// TwinCAT 3 PLC project Recipe_Tool
// ProgramVersion: 3.1.0.8
// libraries:
//   Tc2_Standard, * (Beckhoff Automation GmbH)
//   Tc2_System, * (Beckhoff Automation GmbH)
//   Tc3_Interfaces, * (Beckhoff Automation GmbH)
//   Tc3_Module, * (Beckhoff Automation GmbH)
//   Tc3_PLCopen_OpcUa,3.1.1.0,Beckhoff Automation GmbH
//   UML Statechart Types,4.0.0.0,3S - Smart Software Solutions GmbH
// project tree:
//   DUTs/DUTs/Production List/ DUT_SKILL.TcDUT, DUT_TASK.TcDUT, DUT_TASKSTATE.TcDUT
//   DUTs/DUTs/Queue/ DUT_RECIPEORDER.TcDUT, DUT_RECIPE_USERPARAMETERINPUT.TcDUT
//   DUTs/DUTs/RecipeOffer/ DUT_RECIPEOFFER.TcDUT, DUT_RECIPE_USERPARAMETEROUTPUT.TcDUT
//   DUTs/DUT_BASE/ DUT_PARAMETER_INPUT.TcDUT, DUT_PARAMETER_OUTPUT.TcDUT
//   DUTs/ DUT_MODE.TcDUT, DUT_PARAMETER.TcDUT, DUT_RecipeCommand.TcDUT, DUT_RecToolRECIPEOFFER.TcDUT, DUT_STATEVALUES.TcDUT
//   DUTs/DUT_SERVER/ DUT_SERVER_MODULE_INTERFACE.TcDUT, DUT_SERVER_MODULE_INTERFACE_INPUT.TcDUT, DUT_SERVER_MODULE_INTERFACE_OUTPUT.TcDUT, DUT_SERVER_PARAMETERARRAY.TcDUT, DUT_SERVER_PARAMETERINPUTARRAY.TcDUT, DUT_SERVER_PARAMETEROUTPUTARRAY.TcDUT, DUT_SERVER_SKILL.TcDUT, DUT_SERVER_SKILLARRAY.TcDUT, DUT_SERVER_SKILLINPUTARRAY.TcDUT, DUT_SERVER_SKILLOUTPUTARRAY.TcDUT, DUT_SERVER_SKILL_INPUT.TcDUT, DUT_SERVER_SKILL_OUTPUT.TcDUT, DUT_SERVER_STATEVALUEARRAY.TcDUT, DUT_SERVER_TASK.TcDUT
//   GVLs/ GVL.TcGVL, I_O_GVL.TcGVL, OPCConstants.TcGVL
//   / PlcTask.TcTTO
//   POUs/ FB_AddSkill.TcPOU, FB_ExecuteRecipe.TcPOU, FB_INIT_RECIPE.TcPOU, MAIN.TcPOU, Testing.TcPOU
//   POUs/OPC/ FB_OPCServerConnect.TcPOU, FB_ReadReset.TcPOU, FB_ReadRecipeTool.TcPOU, FB_ReadQueue.TcPOU, FB_UpdateRecipeTool.TcPOU, FB_WriteOfferlist.TcPOU, FB_WriteReset.TcPOU, FB_WriteTask.TcPOU, FB_WriteQueue.TcPOU
//   POUs/Recipes/ Recipe_10000_BlankRecipe.TcPOU, Recipe_10001_OneRound.TcPOU, Recipe_10019_DoubleCookieSimu.TcPOU, Recipe_10018_TripleCookiemitTopping.TcPOU, Recipe_10030_HandModule.TcPOU, Recipe_10050_PumpTest.TcPOU, Recipe_10010_transportreserve.TcPOU, Recipe_10011_Skill1337.TcPOU, Recipe_10012_Skill1337_1338_1339.TcPOU, Recipe_10015_eineCookiebitte.TcPOU, Recipe_10013_nSchichten.TcPOU, Recipe_10014_nSchichten4skills.TcPOU, Recipe_10016_CookiemitTopping.TcPOU, Recipe_10017_DoubleCookiemitTopping.TcPOU, Recipe_10051_FreePassion.TcPOU, Recipe_10054_FreePassion_special.TcPOU, Recipe_10052_Orangenschorle.TcPOU, Recipe_10053_911Targa.TcPOU, Recipe_10054_Sixteen.TcPOU, Recipe_10055_Summerday.TcPOU, Recipe_10056_ArcturianSunrise.TcPOU, Recipe_10057_GreenFive.TcPOU, Recipe_10059_Pina_Batida_Lemon.TcPOU, Recipe_10058_RedOne.TcPOU, Recipe_10100_Initialisation.TcPOU, Recipe_11015_DoubleChocoCookie.TcPOU, Recipe_11020_TequilaSunrise.TcPOU
// real-time tasks:
//   TASK PlcTask: cycle T#10ms, priority 20, ADS port 350

CONFIGURATION Recipe_Tool
    RESOURCE PLC ON TwinCAT3
        TASK PlcTask(INTERVAL := T#10ms, PRIORITY := 20);
        PROGRAM MAIN WITH PlcTask : MAIN;
        PROGRAM Testing WITH PlcTask : Testing;
    END_RESOURCE
END_CONFIGURATION

// ---- DUTs/DUTs/Production List/DUT_SKILL.TcDUT
///  Skill variables inside DUT_TASK
TYPE DUT_SKILL :
STRUCT
	///Name assigned for the process tool
	AssignedModuleName: STRING(80);
	///ID assigned for the process tool
	AssignedModuleID: UINT;
	///Position assigned for the process tool
	AssignedModulePosition: LREAL;
	///Free to use = TRUE, busy to use =FALSE
	Dummy: BOOL := TRUE;
	///Identification number of the skill
	ID: UINT;
	///Name of the skill
	Name: STRING(80);
	///Range of parameters
	Parameter: ARRAY[0..ParameterCnt] OF DUT_PARAMETER;
END_STRUCT
END_TYPE

// ---- DUTs/DUTs/Production List/DUT_TASK.TcDUT
TYPE DUT_TASK :
STRUCT
	///Name of the Task
	Name: STRING(80);
	///Free to use = TRUE, busy to use =FALSE
	Dummy: BOOL := TRUE;
	///Identification number of the Task
	TaskID: INT;
	///Identification number of the Recipe
	RecipeID: INT;
	///Range of Skill in the TASK
	Skill: ARRAY[0..TaskSkillCnt] OF DUT_SKILL;
	///When occurs the action
	Timestamp: STRING(80);
	///State of the TASK e.g (unassigned, assigned, waitingForSkillReady, inProgress, done, aborted, error)
	State: DUT_TASKSTATE := 0;
END_STRUCT
END_TYPE

// ---- DUTs/DUTs/Production List/DUT_TASKSTATE.TcDUT
TYPE DUT_TASKSTATE :
(
	Unassigned := 0,
	///Assigned := 1,
	WaitingForSkillReady := 1,
	InProgress := 2,
	Done := 3,
	Aborted := 4,
	Error := 5
);
END_TYPE

// ---- DUTs/DUTs/Queue/DUT_RECIPEORDER.TcDUT
TYPE DUT_RECIPEORDER :
STRUCT
	Locked: BOOL;
	Pending: BOOL;
	///corelating to the offered recipes#
	RecipeID: INT;
	///continious numbering
	TaskID: INT;
	Name: STRING(80);
	Description: STRING(255);
	UserParameter: ARRAY[0..UserParameterCnt] OF DUT_RECIPE_USERPARAMETERINPUT;
END_STRUCT
END_TYPE

// ---- DUTs/DUTs/Queue/DUT_RECIPE_USERPARAMETERINPUT.TcDUT
TYPE DUT_RECIPE_USERPARAMETERINPUT :
STRUCT
	Value: REAL;
END_STRUCT
END_TYPE

// ---- DUTs/DUTs/RecipeOffer/DUT_RECIPEOFFER.TcDUT
TYPE DUT_RECIPEOFFER :
STRUCT
	Dummy: BOOL := TRUE;
	Name: STRING(80) := 'e.g. Product x';
	RecipeID: INT;
	Description: STRING(255) := '%Description of the Recipe e.g. "a recipe, that produces a product with feature x"';
	UserParameter: ARRAY[0..UserParameterCnt] OF DUT_RECIPE_USERPARAMETEROUTPUT;
END_STRUCT
END_TYPE

// ---- DUTs/DUTs/RecipeOffer/DUT_RECIPE_USERPARAMETEROUTPUT.TcDUT
TYPE DUT_RECIPE_USERPARAMETEROUTPUT :
STRUCT
	Dummy: BOOL := TRUE;
	Name: STRING(80);
	Description: STRING(80);
	Unit: STRING(80);
	MinValue: LREAL;
	MaxValue: LREAL;
	Default: LREAL;
	Step: LREAL;
END_STRUCT
END_TYPE

// ---- DUTs/DUT_BASE/DUT_PARAMETER_INPUT.TcDUT
TYPE DUT_PARAMETER_INPUT :
STRUCT
	///Value of the parameter 
	Value: LREAL;
	///Possibility to a string value depending on the parameter
	StringValue: STRING[80];
END_STRUCT
END_TYPE

// ---- DUTs/DUT_BASE/DUT_PARAMETER_OUTPUT.TcDUT
TYPE DUT_PARAMETER_OUTPUT :
STRUCT
	///Free to use = TRUE, busy to use =FALSE
	Dummy: BOOL := TRUE;
	///ID of the parameter
	ID: UINT;
	///Name of the parameter
	Name: STRING[80];
	///Unit of the parameter
	Unit: STRING[80];
	///Optional parameter
	Required: BOOL;
	///Default parameter to work
	Default: LREAL;
	///Minimum value of the parameter
	MinValue: LREAL;
	///Maximum value of the parameter
	MaxValue: LREAL;
END_STRUCT
END_TYPE

// ---- DUTs/DUT_MODE.TcDUT
/// MODE to run (inside of MODULE_INTERFACE_INPUT)
TYPE DUT_MODE :
(
	///Initialitzation number mode
	Init := 0,
	///Automatic number mode
	Auto := 1,
	///Manual number mode
	Manual := 2,
	Reset := 3
);
END_TYPE

// ---- DUTs/DUT_PARAMETER.TcDUT
TYPE DUT_PARAMETER :
STRUCT
	///Free to use = TRUE, busy to use =FALSE
	Dummy: BOOL := TRUE;
	///ID of the parameter
	ID: UINT;
	///Name of the parameter
	Name: STRING[80];
	///Unit of the parameter (mm,L,...)
	Unit: STRING[80];
	///Optional parameter
	Required: BOOL;
	///Default parameter to work
	Default: LREAL;
	///Minimum value of the parameter
	MinValue: LREAL;
	///Maximum value of the parameter
	MaxValue: LREAL;
	///Actual Value
	Value: LREAL;
	///StringValue
	StringValue: STRING[80];
END_STRUCT
END_TYPE

// ---- DUTs/DUT_RecipeCommand.TcDUT
TYPE DUT_RecipeCommand :
STRUCT
	SkillID: INT;
	SkillName: STRING(80);
	Quantity: LREAL;
END_STRUCT
END_TYPE

// ---- DUTs/DUT_RecToolRECIPEOFFER.TcDUT
TYPE DUT_RecToolRECIPEOFFER :
STRUCT
	Dummy:			BOOL := TRUE;
	Name:			STRING[80]:= 'e.g. Product x';
	RecipeID:		INT;
	Description:	STRING[80]:= '%Description of the Recipe e.g. "a recipe, that produces a product with feature x"';
	UserParameter:  DUT_RECIPE_USERPARAMETEROUTPUT;
END_STRUCT
END_TYPE

// ---- DUTs/DUT_SERVER/DUT_SERVER_MODULE_INTERFACE.TcDUT
/// MODULE INTERFACE INPUT AND OUTPUT 
TYPE DUT_SERVER_MODULE_INTERFACE :
STRUCT
	///Information that the module reads
	Input: DUT_SERVER_MODULE_INTERFACE_INPUT;
	///Information that the module write
	Output: DUT_SERVER_MODULE_INTERFACE_OUTPUT;
END_STRUCT
END_TYPE

// ---- DUTs/DUT_SERVER/DUT_SERVER_MODULE_INTERFACE_INPUT.TcDUT
TYPE DUT_SERVER_MODULE_INTERFACE_INPUT :
STRUCT
	///Mode to run (init,auto,manual,..)
	Mode: DUT_MODE;
	///check if the modules is alive
	ConnectionTestInput: BOOL;
	///Modules get their position
	PositionInput: LREAL;
	///Update data= TRUE, No updatedata=FALSE
	Watchbit: BOOL;
	///Emergency stop
	EmergencyStop: BOOL;
	///Range of INPUT skills
	SkillInput: DUT_SERVER_SKILLINPUTARRAY;
END_STRUCT
END_TYPE

// ---- DUTs/DUT_SERVER/DUT_SERVER_MODULE_INTERFACE_OUTPUT.TcDUT
TYPE DUT_SERVER_MODULE_INTERFACE_OUTPUT :
STRUCT
	///Free to use = TRUE, busy to use =FALSE
	Dummy: BOOL := TRUE;
	///Individual name of the module
	Name: STRING[80];
	///Identification number of module
	ID: UINT;
	///IP address
	IP: STRING[80];
	///Show if the module is in Standby or not
	Idle: BOOL;
	///Show if the module is connected
	Connected: BOOL;
	///Feedback with conection test input
	ConnectionTestOutput: BOOL;
	///Show if the system has error when=TRUE
	Error: BOOL;
	///Identification number of the error
	ErrorID: UINT;
	///Description of the error
	ErrorDescription: STRING[80];
	///Description of the current task
	CurrentTaskDescription: STRING[80];
	///Position of the sensor
	PositionSensor: BOOL;
	///Range of OUTPUT skills
	SkillOutput: DUT_SERVER_SKILLOUTPUTARRAY;
	///Range of state values
	StateValue: DUT_SERVER_STATEVALUEARRAY;
END_STRUCT
END_TYPE

// ---- DUTs/DUT_SERVER/DUT_SERVER_PARAMETERARRAY.TcDUT
TYPE DUT_SERVER_PARAMETERARRAY :
STRUCT
	Parameter0 : DUT_PARAMETER;
	Parameter1 : DUT_PARAMETER;
	Parameter2 : DUT_PARAMETER;
	Parameter3 : DUT_PARAMETER;
	Parameter4 : DUT_PARAMETER;
	Parameter5 : DUT_PARAMETER;
	
END_STRUCT
END_TYPE

// ---- DUTs/DUT_SERVER/DUT_SERVER_PARAMETERINPUTARRAY.TcDUT
TYPE DUT_SERVER_PARAMETERINPUTARRAY :
STRUCT
		Parameterinput0	: DUT_PARAMETER_INPUT;
	Parameterinput1	: DUT_PARAMETER_INPUT;
	Parameterinput2	: DUT_PARAMETER_INPUT;
	Parameterinput3	: DUT_PARAMETER_INPUT;
	Parameterinput4	: DUT_PARAMETER_INPUT;
	Parameterinput5	: DUT_PARAMETER_INPUT;
END_STRUCT
END_TYPE

// ---- DUTs/DUT_SERVER/DUT_SERVER_PARAMETEROUTPUTARRAY.TcDUT
TYPE DUT_SERVER_PARAMETEROUTPUTARRAY :
STRUCT
	ParameterOutput0	: DUT_PARAMETER_OUTPUT;
	ParameterOutput1	: DUT_PARAMETER_OUTPUT;
	ParameterOutput2	: DUT_PARAMETER_OUTPUT;
	ParameterOutput3	: DUT_PARAMETER_OUTPUT;
	ParameterOutput4	: DUT_PARAMETER_OUTPUT;
	ParameterOutput5	: DUT_PARAMETER_OUTPUT;
END_STRUCT
END_TYPE

// ---- DUTs/DUT_SERVER/DUT_SERVER_SKILL.TcDUT
///  Skill variables inside DUT_TASK
TYPE DUT_SERVER_SKILL :
STRUCT
	///Name assigned for the process tool
	AssignedModuleName: STRING[80];
	///ID assigned for the process tool
	AssignedModuleID: UINT;
	///Position assigned for the process tool
	AssignedModulePosition: UINT;
	///Free to use = TRUE, busy to use =FALSE
	Dummy: BOOL := TRUE;
	///Identification number of the skill
	ID: UINT;
	///Name of the skill
	Name: STRING[80];
	///Range of parameters
	Parameter : DUT_SERVER_PARAMETERARRAY;
END_STRUCT
END_TYPE

// ---- DUTs/DUT_SERVER/DUT_SERVER_SKILLARRAY.TcDUT
TYPE DUT_SERVER_SKILLARRAY :
STRUCT
	Skill0 : DUT_SERVER_SKILL;
	Skill1 : DUT_SERVER_SKILL;
	Skill2 : DUT_SERVER_SKILL;
	Skill3 : DUT_SERVER_SKILL;
	Skill4 : DUT_SERVER_SKILL;
	Skill5 : DUT_SERVER_SKILL;
	Skill6 : DUT_SERVER_SKILL;
	Skill7 : DUT_SERVER_SKILL;
	Skill8 : DUT_SERVER_SKILL;
	Skill9 : DUT_SERVER_SKILL;
	Skill10 : DUT_SERVER_SKILL;
	Skill11 : DUT_SERVER_SKILL;
	Skill12 : DUT_SERVER_SKILL;
	Skill13 : DUT_SERVER_SKILL;
	Skill14 : DUT_SERVER_SKILL;
	Skill15 : DUT_SERVER_SKILL;
	Skill16 : DUT_SERVER_SKILL;
	Skill17 : DUT_SERVER_SKILL;
	Skill18 : DUT_SERVER_SKILL;
	Skill19 : DUT_SERVER_SKILL;	
	Skill20 : DUT_SERVER_SKILL;
	Skill21 : DUT_SERVER_SKILL;
	Skill22 : DUT_SERVER_SKILL;
	Skill23 : DUT_SERVER_SKILL;
	Skill24 : DUT_SERVER_SKILL;
	Skill25 : DUT_SERVER_SKILL;
	Skill26 : DUT_SERVER_SKILL;
	Skill27 : DUT_SERVER_SKILL;
	Skill28 : DUT_SERVER_SKILL;
	Skill29 : DUT_SERVER_SKILL;
	Skill30 : DUT_SERVER_SKILL;
	Skill31 : DUT_SERVER_SKILL;
	Skill32 : DUT_SERVER_SKILL;
	Skill33 : DUT_SERVER_SKILL;
	Skill34 : DUT_SERVER_SKILL;
	Skill35 : DUT_SERVER_SKILL;
	Skill36 : DUT_SERVER_SKILL;
	Skill37 : DUT_SERVER_SKILL;
	Skill38 : DUT_SERVER_SKILL;
	Skill39 : DUT_SERVER_SKILL;
	Skill40 : DUT_SERVER_SKILL;
	Skill41 : DUT_SERVER_SKILL;
	Skill42 : DUT_SERVER_SKILL;
	Skill43 : DUT_SERVER_SKILL;
	Skill44 : DUT_SERVER_SKILL;
	Skill45 : DUT_SERVER_SKILL;
	Skill46 : DUT_SERVER_SKILL;
	Skill47 : DUT_SERVER_SKILL;
	Skill48 : DUT_SERVER_SKILL;
	Skill49 : DUT_SERVER_SKILL;
	Skill50 : DUT_SERVER_SKILL;
END_STRUCT
END_TYPE

// ---- DUTs/DUT_SERVER/DUT_SERVER_SKILLINPUTARRAY.TcDUT
TYPE DUT_SERVER_SKILLINPUTARRAY :
STRUCT
	SkillInput0 : DUT_SERVER_SKILL_INPUT;
	SkillInput1 : DUT_SERVER_SKILL_INPUT;
	SkillInput2 : DUT_SERVER_SKILL_INPUT;
	SkillInput3 : DUT_SERVER_SKILL_INPUT;
	SkillInput4 : DUT_SERVER_SKILL_INPUT;
	SkillInput5 : DUT_SERVER_SKILL_INPUT;
	SkillInput6 : DUT_SERVER_SKILL_INPUT;
	SkillInput7 : DUT_SERVER_SKILL_INPUT;
	SkillInput8 : DUT_SERVER_SKILL_INPUT;
	SkillInput9 : DUT_SERVER_SKILL_INPUT;
	SkillInput10 : DUT_SERVER_SKILL_INPUT;
	SkillInput11 : DUT_SERVER_SKILL_INPUT;
	SkillInput12 : DUT_SERVER_SKILL_INPUT;
	SkillInput13 : DUT_SERVER_SKILL_INPUT;
	SkillInput14 : DUT_SERVER_SKILL_INPUT;
	SkillInput15 : DUT_SERVER_SKILL_INPUT;
END_STRUCT
END_TYPE

// ---- DUTs/DUT_SERVER/DUT_SERVER_SKILLOUTPUTARRAY.TcDUT
TYPE DUT_SERVER_SKILLOUTPUTARRAY :
STRUCT
		SkillOutput0	: DUT_SERVER_SKILL_OUTPUT;
	SkillOutput1	: DUT_SERVER_SKILL_OUTPUT;
	SkillOutput2	: DUT_SERVER_SKILL_OUTPUT;
	SkillOutput3	: DUT_SERVER_SKILL_OUTPUT;
	SkillOutput4	: DUT_SERVER_SKILL_OUTPUT;
	SkillOutput5	: DUT_SERVER_SKILL_OUTPUT;
	SkillOutput6	: DUT_SERVER_SKILL_OUTPUT;
	SkillOutput7	: DUT_SERVER_SKILL_OUTPUT;
	SkillOutput8	: DUT_SERVER_SKILL_OUTPUT;
	SkillOutput9	: DUT_SERVER_SKILL_OUTPUT;
	SkillOutput10	: DUT_SERVER_SKILL_OUTPUT;
	SkillOutput11	: DUT_SERVER_SKILL_OUTPUT;
	SkillOutput12	: DUT_SERVER_SKILL_OUTPUT;
	SkillOutput13	: DUT_SERVER_SKILL_OUTPUT;
	SkillOutput14	: DUT_SERVER_SKILL_OUTPUT;
	SkillOutput15	: DUT_SERVER_SKILL_OUTPUT;
END_STRUCT
END_TYPE

// ---- DUTs/DUT_SERVER/DUT_SERVER_SKILL_INPUT.TcDUT
TYPE DUT_SERVER_SKILL_INPUT :
STRUCT
	///Range of parameters
	ParameterInput: DUT_SERVER_PARAMETERINPUTARRAY;
	///Start process
	Execute: BOOL;
END_STRUCT
END_TYPE

// ---- DUTs/DUT_SERVER/DUT_SERVER_SKILL_OUTPUT.TcDUT
TYPE DUT_SERVER_SKILL_OUTPUT :
STRUCT
	///Free to use = TRUE, busy to use =FALSE
	Dummy: BOOL := TRUE;
	///Identification number of skill
	ID: UINT;
	///indentfication name of skill
	Name: STRING[80];
	///Skill activated
	Activated: BOOL;
	///Ready to do skill
	Ready: BOOL;
	///Skill in process
	Busy: BOOL;
	///Skill finish
	Done: BOOL;
	///Error in system
	Error: BOOL;
	///Range of parameters
	ParameterOutput: DUT_SERVER_PARAMETEROUTPUTARRAY;
END_STRUCT
END_TYPE

// ---- DUTs/DUT_SERVER/DUT_SERVER_STATEVALUEARRAY.TcDUT
TYPE DUT_SERVER_STATEVALUEARRAY :
STRUCT
		Statevalue0	: DUT_STATEVALUES;
	Statevalue1	: DUT_STATEVALUES;
	Statevalue2	: DUT_STATEVALUES;
	Statevalue3	: DUT_STATEVALUES;
	Statevalue4	: DUT_STATEVALUES;
	Statevalue5	: DUT_STATEVALUES;
	Statevalue6	: DUT_STATEVALUES;
	Statevalue7	: DUT_STATEVALUES;
	Statevalue8	: DUT_STATEVALUES;
	Statevalue9	: DUT_STATEVALUES;
	Statevalue10	: DUT_STATEVALUES;
END_STRUCT
END_TYPE

// ---- DUTs/DUT_SERVER/DUT_SERVER_TASK.TcDUT
TYPE DUT_SERVER_TASK :
STRUCT
	///Name of the Task
	Name: STRING[80];
	///Free to use = TRUE, busy to use =FALSE
	Dummy: BOOL := TRUE;
	///Identification number of the Task
	TaskID: INT;
	///Identification number of the Recipe
	RecipeID: INT;
	///Range of Skill in the TASK
	Skill: DUT_SERVER_SKILLARRAY;
	///When occurs the action
	Timestamp: STRING[80];
	///State of the TASK e.g (unassigned, assigned, waitingForSkillReady, inProgress, done, aborted, error)
	State: DUT_TASKSTATE;
END_STRUCT
END_TYPE

// ---- DUTs/DUT_STATEVALUES.TcDUT
TYPE DUT_STATEVALUES :
STRUCT
	Dummy:			BOOL := TRUE;				(*Free to use = TRUE, busy to use =FALSE*)
	Value:			LREAL;						(*Value of the State*)
	Name:			STRING[80];						(*Name of the state*)
	Description:	STRING[80];				(*Description of the state*)
	Unit:			STRING[80];						(*Unit of the state ()*)
END_STRUCT
END_TYPE

// ---- GVLs/GVL.TcGVL
VAR_GLOBAL
	ExecuteSkill	: FB_AddSkill;
	TempTask		: DUT_TASK;
	EmptyTask		: DUT_TASK;
	EmptyQueue		: DUT_RECIPEORDER;
	
	ZCremeModuleCalibration		: LREAL := 0;	
	ZCremeModule				: LREAL	:= 101;
	
	
	ZCocktailModuleCalibration 	: LREAL := 0;
	ZCocktailModule				: LREAL := 20;
	
	ZCookieModuleCalibration	: LREAL := 0;
	ZCookieModule				: LREAL := 90.0;
	
	ZInputOutput				: LREAL := 109;
	
	
	
	cookiethickness				: LREAL := 5.0;
	toppingthickness			: LREAL := 1.0;
	
	preasureheight				: LREAL := 30.0;
	ClearTaskList				: BOOL;	
	ClearManual					: BOOL;
END_VAR

// ---- GVLs/I_O_GVL.TcGVL
VAR_GLOBAL
// Inputs:

Queue	: DUT_RECIPEORDER;

//Outputs:

Offer	: ARRAY [0..OfferCnt] OF DUT_RECIPEOFFER;

// ProductionList

Task	: ARRAY [0..TaskCnt] OF DUT_TASK;
END_VAR

// ---- GVLs/OPCConstants.TcGVL
VAR_GLOBAL CONSTANT
	///Maximum number of skillparameters:
	ParameterCnt: INT := 5;
	///Maximum number of skills per Module:
	SkillCnt: INT := 15;
	///Maximum number of Statevalues of one Module:
	StateCnt: INT := 10;
	///Maximum number of modules:
	ModuleCnt: INT := 10;
	///Maximum number of Tasks in Production List:
	TaskCnt: INT := 30;
	///Maximum number  of offered recipes:
	OfferCnt: INT := 30;
	///Maximum number of Orders in Queue:
	OrderCnt: INT := 5;
	///Number of user set parameters per recipe:
	UserParameterCnt: INT := 5;
	///Number of skills per task:
	TaskSkillCnt: INT := 50;
	
	
END_VAR

// ---- POUs/MAIN.TcPOU
PROGRAM MAIN
VAR
	
		
	state	: INT := -40;	
	i		: INT;
	connectcounter	: INT;
	TaskListPosition: INT := -1;
	TaskListPositionString	: STRING[80];
	Tempstring		: STRING[80];
	//FB Instances
	TranslateRecipe	: FB_ExecuteRecipe;
	fbInitOffers	: FB_INIT_RECIPE;	
	//OPC Instances:
	//fbOPCUpdate		: FB_UpdateRecipeTool;
	fbReadReset			: FB_ReadReset;
	fbWriteReset		: FB_WriteReset;
	fbOPCConnect		: FB_OPCServerConnect;
	fbWriteOffers		: FB_WriteOfferlist;
	fbReadQueue			: FB_ReadQueue;
	fbWriteTask			: FB_WriteTask;
	fbWriteQueue		: FB_WriteQueue;
	fbDisconnect		: UA_Disconnect;
	NamespaceIndex		: UINT;
	ConnectionHdl		: DWORD;
	TaskIdentifier		: STRING[80];
	sizeofRecipfOFfer	: INT;
	ClearOrder			: DUT_RECIPEORDER;
	ToolTimeout			: TON;
	Trigger				: R_TRIG;
	TriggerState		: INT;
	ResetReadTimer		: TON;
	
END_VAR


CASE state OF
	-40: //Initialate Recipe Offer List
		fbInitOffers(Execute := TRUE);
		ToolTimeout(IN := FALSE);
		IF fbInitOffers.Done THEN
			state := -30;
		END_IF
	-35: fbDisconnect(ConnectionHdl := ConnectionHdl,Timeout := T#4S, Execute := FALSE);
		state := -34;
	-34: fbDisconnect(ConnectionHdl := ConnectionHdl,Timeout := T#4s, Execute := TRUE);
		IF nOT fbDisconnect.busy  THEN
			state := -30;
		END_IF
		
	
	-30: fbOPCConnect(
						ServerUrl:= 'opc.tcp://192.168.42.42:4840',//'opc.tcp://192.168.192.116:4840', 
						NamespaceUri:= 'PLC1', 
						ClientName:= 'RecipeTool', 
						execute:= TRUE, 
						ConnectHdl=> ConnectionHdl, 
						Namespaceindex=> NamespaceIndex, 
						busy=> , 
						done=> , 
						error=> );
		IF fbOPCConnect.done THEN
			state := -15;
		END_IF
					
		
	
	
	
	-15: // OPC WRITE 
		fbWriteOffers(
						WriteIdentifier:= 'MI5.Recipe', 
						NamespaceIndex:= NamespaceIndex, 
						ConnectionHdl:= ConnectionHdl, 
						execute:= TRUE, 
						WriteData:= Offer, 
						done=> , 
						busy=> , 
						error=> );
		IF fbWriteOffers.done THEN
			state := -10;
		END_IF

	
	-10: //INIT DONE
		TranslateRecipe.InitDone := TRUE;
		state := 0;
	
	
	
	 0:		// Waiting for new Order
	 	IF NOT Testing.NoOPC THEN
	 		fbReadQueue(
						ReadIdentifier:= 'MI5.Order[0]', 
						NamespaceIndex:= NamespaceIndex, 
						ConnectionHdl:= ConnectionHdl, 
						execute:= TRUE, 
						ReadData=> Queue, 
						done=> , 
						busy=> , 
						error=> );
			IF fbReadQueue.done THEN
				state := 1;
			END_IF
		ELSE
			state := 5;
		END_IF
		
	1:	
		IF NOT Testing.NoOPC THEN
				fbReadQueue(
							ReadIdentifier:= 'MI5.Order[0]', 
							NamespaceIndex:= NamespaceIndex, 
							ConnectionHdl:= ConnectionHdl, 
							execute:= TRUE, 
							ReadData=> Queue, 
							done=> , 
							busy=> , 
							error=> );
				Trigger(CLK := fbReadQueue.done);
				ToolTimeout(IN := NOT Trigger.Q);
							
				IF Queue.Pending THEN
					state := 10;
					TaskListPosition := TaskListPosition +1;
						//Reset bei Overflow
						IF TaskListPosition > 29 THEN
							TaskListPosition := 0;
						END_IF
				END_IF		
		ELSE
			state := 5;
		END_IF
	 5:
		IF Queue.Pending THEN
			state := 10;
			TaskListPosition := TaskListPosition +1;
				//Reset bei Overflow
				IF TaskListPosition > 29 THEN
					TaskListPosition := 0;
				END_IF
		END_IF
	 	
	 
	10: state := 20;
		
		
	20: //Translate corresponding offer to TempTask
		TranslateRecipe(Order:= Queue, Done=> , Execute := TRUE);
		
		IF TranslateRecipe.Done THEN
			state := 21;//21;
			ExecuteSkill.TargetSkillNo := 0;
		END_IF
		
		
		//todo quatsch recipe IDs abfangen? return an HMI
	21: TempTask.Name := Queue.Name;
		TempTask.Dummy := FALSE;
		TempTask.RecipeID := Queue.RecipeID;
		TempTask.TaskID := Queue.TaskID;
		TempTask.State := 1;
		TempTask.Timestamp := 'mytimestamp';
		state := 25;
		
			
	25: //Parse write identifier
		TaskListPositionString := INT_TO_STRING(TaskListPosition);
		Tempstring := CONCAT(STR1:= 'MI5.ProductionList[', STR2:= TaskListPositionString );
		
		TaskIdentifier := CONCAT(STR1:= Tempstring, STR2:=']' );
		state := 30;	
	30: // Copy to local Production List
		fbWriteTask(
					WriteIdentifier:= TaskIdentifier, 
					NamespaceIndex:= NamespaceIndex, 
					ConnectionHdl:= ConnectionHdl, 
					execute:= TRUE, 
					WriteData:= TempTask, 
					done=> , 
					busy=> , 
					error=> );
		IF fbWriteTask.done THEN
		//
		state := 40;
		END_IF		
	

	40:  // free Queue Slot
		TempTask				:= EmptyTask;
		IF NOT Testing.NoOPC THEN
			fbWriteQueue(
				WriteIdentifier:= 'MI5.Order[0]', 
				NamespaceIndex:= NamespaceIndex, 
				ConnectionHdl:= ConnectionHdl, 
				execute:= TRUE, 
				WriteData:= , 
				done=> , 
				busy=> , 
				error=> );
			IF fbWriteQueue.done THEN
			state := 0;
			END_IF
		ELSE
			Queue.Pending := FALSE;
			state := 0;
		END_IF
	
	
		
		
		
	125: //Parse write identifier
		TaskListPositionString := INT_TO_STRING(i);
		Tempstring := CONCAT(STR1:= 'MI5.ProductionList[', STR2:= TaskListPositionString );
		
		TaskIdentifier := CONCAT(STR1:= Tempstring, STR2:=']' );
		state := 130;	
	130: // Copy to local Production List
		fbWriteTask(
					WriteIdentifier:= TaskIdentifier, 
					NamespaceIndex:= NamespaceIndex, 
					ConnectionHdl:= ConnectionHdl, 
					execute:= TRUE, 
					WriteData:= EmptyTask, 
					done=> , 
					busy=> , 
					error=> );
		IF fbWriteTask.done THEN
			IF  i <TaskCnt  THEN
				i := i +1;
				state := 125;
			ELSE
				state := -30;
				i := -1;
			END_IF
		
		END_IF		
		
		
END_CASE



sizeofRecipfOFfer := SIZEOF(DUT_RecipeOffer);

//TImerout:
ToolTimeout(IN := TRUE, PT := T#20S);


//stateänderungsüberprüfung
IF NOT (state  = triggerstate) THEN
	ToolTimeout(IN:= FALSE);
END_IF
triggerstate := state;


IF ToolTimeout.Q THEN
	connectcounter	:= connectcounter +1;
	state := -35;
	ToolTimeout(IN:= FALSE);
	fbOPCConnect	(execute := FALSE);			
	fbWriteOffers	(execute := FALSE);		
	fbReadQueue		(execute := FALSE);			
	fbWriteTask		(execute := FALSE);			
	fbWriteQueue	(execute := FALSE);		
	
END_IF

ResetReadTimer(IN := TRUE, PT := T#3S);
IF ResetReadTimer.Q THEN
	ResetReadTimer(IN := FALSE);
	ResetReadTimer(IN := TRUE);
	fbReadReset.execute := TRUE;
END_IF
fbReadReset(		ReadIdentifier:= 'MI5.ClearTaskList', 
					NamespaceIndex:= NamespaceIndex, 
					ConnectionHdl:= ConnectionHdl, 
					execute:= , 
					ReadData=> ClearTaskList, 
					done=> , 
					busy=> , 
					error=> 
				);

					
IF ClearTaskList OR ClearManual THEN
	i := 0;
	ClearManual := FALSE;
	Tasklistposition := -1;
	fbWriteReset(	WriteIdentifier := 'MI5.ClearTaskList',
					NamespaceIndex := NamespaceIndex, 
					ConnectionHdl := ConnectionHdl, 
					WriteData := FALSE,
					Execute		:= TRUE);
	IF fbWriteReset.done THEN
		state := 125;
	END_IF
	
END_IF

END_PROGRAM

// ---- POUs/FB_ExecuteRecipe.TcPOU
FUNCTION_BLOCK FB_ExecuteRecipe
VAR_INPUT
	Order			: 	DUT_RECIPEORDER;
	Execute			: 	BOOL;
	InitDone		: 	BOOL;
END_VAR
VAR_OUTPUT
	Done	:	BOOL;
	NotAvailable: BOOL;
	RecipeInfo	: DUT_RECIPEOFFER;
END_VAR
VAR
		BriefcaseConfig	: BOOL := TRUE;
		i			: INT;
		Recipe10001 : Recipe_10001_OneRound;
		Recipe10010 : Recipe_10010_transportreserve;
		
		
		//Recipe11020	: Recipe_11020_TequilaSunrise;
		Recipe10000 : Recipe_10000_BlankRecipe;
		//Recipe10013 : Recipe_10013_nSchichten;
		//Recipe10014 : Recipe_10014_nSchichten4skills;
		//Recipe20014	: Recipe_20014_chocoCookie;
		Recipe10011: Recipe_10011_Skill1337;
		//Recipe10012: Recipe_10012_Skill1337_1338_1339;
		//Recipe10015: Recipe_10015_eineCookiebitte;
		//Recipe10016: Recipe_10016_CookiemitTopping;
		Recipe10017: Recipe_10017_DoubleCookiemitTopping;
		//Recipe10018: Recipe_10018_TripleCookiemitTopping;
		Recipe10019: Recipe_10019_DoubleCookieSimu;
		//Recipe10050: Recipe_10050_PumpTest;
		Recipe10051: Recipe_10051_FreePassion;
		//Recipe10052: Recipe_10052_Orangenschorle;
		Recipe10053: Recipe_10053_911Targa;
		//Recipe10054: Recipe_10054_FreePassion_special;
		Recipe10055: Recipe_10055_Summerday;
		Recipe10056: Recipe_10056_ArcturianSunrise;
		Recipe10057: Recipe_10057_GreenFive;
		//Recipe10058: Recipe_10058_RedOne;
		//Recipe10059: Recipe_10059_Pina_Batida_Lemon;
		
END_VAR





IF Execute THEN
	Done := FALSE;
	NotAvailable := FALSE;
	
	CASE Order.RecipeID OF
		
		(*10000: Recipe10000 (Execute := InitDone,Order := order,RecipeInfo => RecipeInfo);
				
				IF Recipe10000.RecipeDone THEN
					Done := TRUE;
					Execute := FALSE;
					Recipe10000(execute := FALSE);
					
					
				END_IF
		*)		
		
		10001: Recipe10001 (Execute := InitDone,Order := order,RecipeInfo => RecipeInfo);
				
				IF Recipe10001.RecipeDone THEN
					Done := TRUE;
					Execute := FALSE;
					Recipe10001(execute := FALSE);
										
				END_IF	
				
		10010: Recipe10010 (Execute := InitDone,Order := order,RecipeInfo => RecipeInfo);
				
				IF Recipe10010.RecipeDone THEN
					Done := TRUE;
					Execute := FALSE;
					Recipe10010(execute := FALSE);
										
				END_IF
		10011: Recipe10011 (Execute := InitDone,Order := order,RecipeInfo => RecipeInfo);
				
				IF Recipe10011.RecipeDone THEN
					Done := TRUE;
					Execute := FALSE;
					Recipe10011(execute := FALSE);
										
				END_IF
				
		(*10012: Recipe10012 (Execute := InitDone,Order := order,RecipeInfo => RecipeInfo);
				
				IF Recipe10012.RecipeDone THEN
					Done := TRUE;
					Execute := FALSE;
					Recipe10012(execute := FALSE);
										
				END_IF
		*)
		(*
10013: Recipe10013 (Execute := InitDone,Order := order,RecipeInfo => RecipeInfo);
				
				IF Recipe10013.RecipeDone THEN
					Done := TRUE;
					Execute := FALSE;
					Recipe10013(execute := FALSE);
										
				END_IF
				*)
		(*10014: Recipe10014 (Execute := InitDone,Order := order,RecipeInfo => RecipeInfo);
				
				IF Recipe10014.RecipeDone THEN
					Done := TRUE;
					Execute := FALSE;
					Recipe10014(execute := FALSE);
										
				END_IF*)
		(*10015: Recipe10015 (Execute := InitDone,Order := order,RecipeInfo => RecipeInfo);
				
				IF Recipe10015.RecipeDone THEN
					Done := TRUE;
					Execute := FALSE;
					Recipe10015(execute := FALSE);
										
				END_IF
		*)
		
		(*
		10016: Recipe10016 (Execute := InitDone,Order := order,RecipeInfo => RecipeInfo);
				
				IF Recipe10016.RecipeDone THEN
					Done := TRUE;
					Execute := FALSE;
					Recipe10016(execute := FALSE);
										
				END_IF
				*)
				
		10017: Recipe10017 (Execute := InitDone,Order := order,RecipeInfo => RecipeInfo);
				
				IF Recipe10017.RecipeDone THEN
					Done := TRUE;
					Execute := FALSE;
					Recipe10017(execute := FALSE);
										
				END_IF	
		(*10018: Recipe10018 (Execute := InitDone,Order := order,RecipeInfo => RecipeInfo);
				
				IF Recipe10018.RecipeDone THEN
					Done := TRUE;
					Execute := FALSE;
					Recipe10018(execute := FALSE);
										
				END_IF		
			*)	
		10019: Recipe10019 (Execute := InitDone,Order := order,RecipeInfo => RecipeInfo);
				
				IF Recipe10019.RecipeDone THEN
					Done := TRUE;
					Execute := FALSE;
					Recipe10019(execute := FALSE);
										
				END_IF
		(*10050: Recipe10050 (Execute := InitDone,Order := order,RecipeInfo => RecipeInfo);
				
				IF Recipe10050.RecipeDone THEN
					Done := TRUE;
					Execute := FALSE;
					Recipe10050(execute := FALSE);
										
				END_IF	*)
		
		10051: Recipe10051 (Execute := InitDone,Order := order,RecipeInfo => RecipeInfo);
				
				IF Recipe10051.RecipeDone THEN
					Done := TRUE;
					Execute := FALSE;
					Recipe10051(execute := FALSE);
										
				END_IF	
		
		(*10052: Recipe10052 (Execute := InitDone,Order := order,RecipeInfo => RecipeInfo);
				
				IF Recipe10052.RecipeDone THEN
					Done := TRUE;
					Execute := FALSE;
					Recipe10052(execute := FALSE);
										
				END_IF*)
		
		10053: Recipe10053 (Execute := InitDone,Order := order,RecipeInfo => RecipeInfo);
				
				IF Recipe10053.RecipeDone THEN
					Done := TRUE;
					Execute := FALSE;
					Recipe10053(execute := FALSE);
										
				END_IF		
				
		(*10054: Recipe10054 (Execute := InitDone,Order := order,RecipeInfo => RecipeInfo);
				
				IF Recipe10054.RecipeDone THEN
					Done := TRUE;
					Execute := FALSE;
					Recipe10054(execute := FALSE);
										
				END_IF			
				*)
		10055: 
				IF NOT BriefcaseConfig THEN
			   		Recipe10055 (Execute := InitDone,Order := order,RecipeInfo => RecipeInfo);
				
					IF Recipe10055.RecipeDone THEN
						Done := TRUE;
						Execute := FALSE;
						Recipe10055(execute := FALSE);
											
					END_IF	
				ELSE
					Done := TRUE;
					NotAvailable := TRUE;
					Execute := FALSE;
				END_IF		
				
		10056: IF NOT BriefcaseConfig THEN
			   		Recipe10056 (Execute := InitDone,Order := order,RecipeInfo => RecipeInfo);
				
					IF Recipe10056.RecipeDone THEN
						Done := TRUE;
						Execute := FALSE;
						Recipe10056(execute := FALSE);
											
					END_IF	
				ELSE
					Done := TRUE;
					NotAvailable := TRUE;
					Execute := FALSE;
				END_IF	
		
				
		10057: IF NOT BriefcaseConfig THEN
			   		Recipe10057 (Execute := InitDone,Order := order,RecipeInfo => RecipeInfo);
				
					IF Recipe10057.RecipeDone THEN
						Done := TRUE;
						Execute := FALSE;
						Recipe10057(execute := FALSE);
											
					END_IF	
				ELSE
					Done := TRUE;
					NotAvailable := TRUE;
					Execute := FALSE;
				END_IF	
		
		
		(*10059: IF NOT BriefcaseConfig THEN
			   		Recipe10059 (Execute := InitDone,Order := order,RecipeInfo => RecipeInfo);
				
					IF Recipe10059.RecipeDone THEN
						Done := TRUE;
						Execute := FALSE;
						Recipe10059(execute := FALSE);
											
					END_IF	
				ELSE
					Done := TRUE;
					NotAvailable := TRUE;
					Execute := FALSE;
				END_IF
				*)
				
				
				
				
				
				
				
		ELSE 
				Done := TRUE;
				NotAvailable := TRUE;
				Execute := FALSE;				
			
	END_CASE
	IF NOT InitDone THEN					
						Done := TRUE;				
						Execute := FALSE;
					
	END_IF
END_IF

END_FUNCTION_BLOCK

// ---- POUs/Recipes/Recipe_10001_OneRound.TcPOU
FUNCTION_BLOCK Recipe_10001_OneRound
VAR_INPUT
	execute	: BOOL;
	Order	: DUT_RECIPEORDER;
END_VAR
VAR_OUTPUT
	RecipeInfo	: DUT_RECIPEOFFER;
	RecipeDone	: BOOL;	
	InitDone	: BOOL;
END_VAR
VAR
	StepDone	: BOOL;
END_VAR

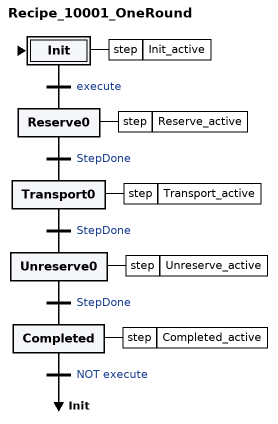
INITIAL_STEP Init:
    Init_active(N);  // step action
END_STEP
TRANSITION FROM Init TO Reserve0
    := execute;
END_TRANSITION
STEP Reserve0:
    Reserve_active(N);  // step action
END_STEP
TRANSITION FROM Reserve0 TO Transport0
    := StepDone;
END_TRANSITION
STEP Transport0:
    Transport_active(N);  // step action
END_STEP
TRANSITION FROM Transport0 TO Unreserve0
    := StepDone;
END_TRANSITION
STEP Unreserve0:
    Unreserve_active(N);  // step action
END_STEP
TRANSITION FROM Unreserve0 TO Completed
    := StepDone;
END_TRANSITION
STEP Completed:
    Completed_active(N);  // step action
END_STEP
TRANSITION FROM Completed TO Init
    := NOT execute;
END_TRANSITION

ACTION Unblock2_active:
StepDone := FALSE;

//Skill auswählen
ExecuteSkill.SkillID 		:= 1316;
ExecuteSkill.SkillName	 	:= 'Unblock';

//Parameter setzen

ExecuteSkill.Parameter[1].ID := 1;
ExecuteSkill.Parameter[1].Name := 'TaskID';
ExecuteSkill.Parameter[1].Value := 131;


(*
ExecuteSkill.Parameter[2].ID := ;
ExecuteSkill.Parameter[2].Name := '';
ExecuteSkill.Parameter[2].Value := ;
*)

(*
ExecuteSkill.Parameter[3].ID := ;
ExecuteSkill.Parameter[3].Name := '';
ExecuteSkill.Parameter[3].Value := ;
*)

(*
ExecuteSkill.Parameter[4].ID := ;
ExecuteSkill.Parameter[4].Name := '';
ExecuteSkill.Parameter[4].Value := ;
*)

(*
ExecuteSkill.Parameter[5].ID := ;
ExecuteSkill.Parameter[5].Name := '';
ExecuteSkill.Parameter[5].Value := ;
*)



ExecuteSkill();

StepDone := ExecuteSkill.Done;
END_ACTION

ACTION Transport1_active:
StepDone := FALSE;

//Skill auswählen
ExecuteSkill.SkillID 		:= 1320;
ExecuteSkill.SkillName	 	:= 'Name';

//Parameter setzen

ExecuteSkill.Parameter[3].ID := 3;
ExecuteSkill.Parameter[3].Name := 'Velocity';
ExecuteSkill.Parameter[3].Value := 2500;



ExecuteSkill.Parameter[4].ID := 4 ;
ExecuteSkill.Parameter[4].Name := 'Acceleration';
ExecuteSkill.Parameter[4].Value := 1000 ;



ExecuteSkill.Parameter[1].ID := 1;
ExecuteSkill.Parameter[1].Name := 'TargetPosition X';
ExecuteSkill.Parameter[1].Value := 3200 ;
ExecuteSkill.Parameter[1].StringValue := '#DP#2#XPosition' ;




ExecuteSkill.Parameter[2].ID := 2;
ExecuteSkill.Parameter[2].Name := 'TargetPosition Z';
ExecuteSkill.Parameter[2].Value := 65 ;


(*
ExecuteSkill.Parameter[5].ID := ;
ExecuteSkill.Parameter[5].Name := '';
ExecuteSkill.Parameter[5].Value := ;
*)



ExecuteSkill();

StepDone := ExecuteSkill.Done;
END_ACTION

ACTION Reserve_active:
StepDone := FALSE;
RecipeDone := FALSE;
//Skill auswählen
ExecuteSkill.SkillID 		:= 1310;
ExecuteSkill.SkillName	 	:= 'Reserve';

//Parameter setzen

ExecuteSkill.Parameter[1].ID := 1;
ExecuteSkill.Parameter[1].Name := 'TaskID';
ExecuteSkill.Parameter[1].Value := 123;


(*
ExecuteSkill.Parameter[2].ID := ;
ExecuteSkill.Parameter[2].Name := '';
ExecuteSkill.Parameter[2].Value := ;
*)

(*
ExecuteSkill.Parameter[3].ID := ;
ExecuteSkill.Parameter[3].Name := '';
ExecuteSkill.Parameter[3].Value := ;
*)

(*
ExecuteSkill.Parameter[4].ID := ;
ExecuteSkill.Parameter[4].Name := '';
ExecuteSkill.Parameter[4].Value := ;
*)

(*
ExecuteSkill.Parameter[5].ID := ;
ExecuteSkill.Parameter[5].Name := '';
ExecuteSkill.Parameter[5].Value := ;
*)



ExecuteSkill();

StepDone := ExecuteSkill.Done;
END_ACTION

ACTION Transport_active:
StepDone := FALSE;

//Skill auswählen
ExecuteSkill.SkillID 		:= 1320;
ExecuteSkill.SkillName	 	:= 'Transport';

//Parameter setzen
ExecuteSkill.Parameter[3].Dummy := FALSE;
ExecuteSkill.Parameter[3].ID :=3 ;
ExecuteSkill.Parameter[3].Name := 'Velocity';
ExecuteSkill.Parameter[3].Value := 3000;


ExecuteSkill.Parameter[1].Dummy := FALSE;
ExecuteSkill.Parameter[1].ID :=1 ;
ExecuteSkill.Parameter[1].Name := 'TargetPosition X';
ExecuteSkill.Parameter[1].Value := 1499.0;


ExecuteSkill.Parameter[2].Dummy := FALSE;
ExecuteSkill.Parameter[2].ID := 2 ;
ExecuteSkill.Parameter[2].Name := 'TargetPosition Z';
ExecuteSkill.Parameter[2].Value := 0 ;


ExecuteSkill.Parameter[4].Dummy := FALSE;
ExecuteSkill.Parameter[4].ID := 4 ;
ExecuteSkill.Parameter[4].Name := 'Acceleration';
ExecuteSkill.Parameter[4].Value := 4000;


(*
ExecuteSkill.Parameter[5].ID := ;
ExecuteSkill.Parameter[5].Name := '';
ExecuteSkill.Parameter[5].Value := ;
*)



ExecuteSkill();

StepDone := ExecuteSkill.Done;
END_ACTION

ACTION Completed_active:
RecipeDone := TRUE;
StepDone := FALSE;
END_ACTION

ACTION Unreserve_active:
StepDone := FALSE;

//Skill auswählen
ExecuteSkill.SkillID 		:= 1311;
ExecuteSkill.SkillName	 	:= 'Unreserve';

//Parameter setzen

ExecuteSkill.Parameter[1].ID := 1;
ExecuteSkill.Parameter[1].Name := 'TaskID';
ExecuteSkill.Parameter[1].Value := 131;


(*
ExecuteSkill.Parameter[2].ID := ;
ExecuteSkill.Parameter[2].Name := '';
ExecuteSkill.Parameter[2].Value := ;
*)

(*
ExecuteSkill.Parameter[3].ID := ;
ExecuteSkill.Parameter[3].Name := '';
ExecuteSkill.Parameter[3].Value := ;
*)

(*
ExecuteSkill.Parameter[4].ID := ;
ExecuteSkill.Parameter[4].Name := '';
ExecuteSkill.Parameter[4].Value := ;
*)

(*
ExecuteSkill.Parameter[5].ID := ;
ExecuteSkill.Parameter[5].Name := '';
ExecuteSkill.Parameter[5].Value := ;
*)



ExecuteSkill();

StepDone := ExecuteSkill.Done;
END_ACTION

ACTION Init_active:
RecipeDone := FALSE;

// Initialisation of Recipe Parameters an name etc
RecipeInfo.Name := 'XTS one Round';
RecipeInfo.Description := 'One Single Transport';
RecipeInfo.Dummy := FALSE;
RecipeInfo.RecipeID := 10001; 	// 
Initdone := TRUE;

//Parameter 1:
(*
	RecipeInfo.UserParameter[1].Dummy 		:= 
	RecipeInfo.UserParameter[1].Default		:=
	RecipeInfo.UserParameter[1].Description	:=
	RecipeInfo.UserParameter[1].MaxValue	:=
	RecipeInfo.UserParameter[1].MinValue	:=
	RecipeInfo.UserParameter[1].Name		:=
	RecipeInfo.UserParameter[1].Unit		:=
*)
//Parameter 2:

(*
	RecipeInfo.UserParameter[2].Dummy 		:= 
	RecipeInfo.UserParameter[2].Default		:=
	RecipeInfo.UserParameter[2].Description	:=
	RecipeInfo.UserParameter[2].MaxValue	:=
	RecipeInfo.UserParameter[2].MinValue	:=
	RecipeInfo.UserParameter[2].Name		:=
	RecipeInfo.UserParameter[2].Unit		:=
*)

//Parameter 3:

(*
	RecipeInfo.UserParameter[3].Dummy 		:= 
	RecipeInfo.UserParameter[3].Default		:=
	RecipeInfo.UserParameter[3].Description	:=
	RecipeInfo.UserParameter[3].MaxValue	:=
	RecipeInfo.UserParameter[3].MinValue	:=
	RecipeInfo.UserParameter[3].Name		:=
	RecipeInfo.UserParameter[3].Unit		:=
*)

//Parameter 4:

(*
	RecipeInfo.UserParameter[4].Dummy 		:= 
	RecipeInfo.UserParameter[4].Default		:=
	RecipeInfo.UserParameter[4].Description	:=
	RecipeInfo.UserParameter[4].MaxValue	:=
	RecipeInfo.UserParameter[4].MinValue	:=
	RecipeInfo.UserParameter[4].Name		:=
	RecipeInfo.UserParameter[4].Unit		:=
*)


//Parameter 5:

(*
	RecipeInfo.UserParameter[5].Dummy 		:= 
	RecipeInfo.UserParameter[5].Default		:=
	RecipeInfo.UserParameter[5].Description	:=
	RecipeInfo.UserParameter[5].MaxValue	:=
	RecipeInfo.UserParameter[5].MinValue	:=
	RecipeInfo.UserParameter[5].Name		:=
	RecipeInfo.UserParameter[5].Unit		:=
*)
END_ACTION

ACTION Unblock1_active:
StepDone := FALSE;

//Skill auswählen
ExecuteSkill.SkillID 		:= 1316;
ExecuteSkill.SkillName	 	:= 'Unblock';

//Parameter setzen

ExecuteSkill.Parameter[1].ID := 1;
ExecuteSkill.Parameter[1].Name := 'TaskID';
ExecuteSkill.Parameter[1].Value := 128 ;


(*
ExecuteSkill.Parameter[2].ID := ;
ExecuteSkill.Parameter[2].Name := '';
ExecuteSkill.Parameter[2].Value := ;
*)

(*
ExecuteSkill.Parameter[3].ID := ;
ExecuteSkill.Parameter[3].Name := '';
ExecuteSkill.Parameter[3].Value := ;
*)

(*
ExecuteSkill.Parameter[4].ID := ;
ExecuteSkill.Parameter[4].Name := '';
ExecuteSkill.Parameter[4].Value := ;
*)

(*
ExecuteSkill.Parameter[5].ID := ;
ExecuteSkill.Parameter[5].Name := '';
ExecuteSkill.Parameter[5].Value := ;
*)



ExecuteSkill();

StepDone := ExecuteSkill.Done;
END_ACTION

ACTION Block2_active:
StepDone := FALSE;

//Skill auswählen
ExecuteSkill.SkillID 		:= 1315;
ExecuteSkill.SkillName	 	:= 'Block';

//Parameter setzen

ExecuteSkill.Parameter[1].ID := 1;
ExecuteSkill.Parameter[1].Name := 'TaskID';
ExecuteSkill.Parameter[1].Value := 130;


(*
ExecuteSkill.Parameter[2].ID := ;
ExecuteSkill.Parameter[2].Name := '';
ExecuteSkill.Parameter[2].Value := ;
*)

(*
ExecuteSkill.Parameter[3].ID := ;
ExecuteSkill.Parameter[3].Name := '';
ExecuteSkill.Parameter[3].Value := ;
*)

(*
ExecuteSkill.Parameter[4].ID := ;
ExecuteSkill.Parameter[4].Name := '';
ExecuteSkill.Parameter[4].Value := ;
*)

(*
ExecuteSkill.Parameter[5].ID := ;
ExecuteSkill.Parameter[5].Name := '';
ExecuteSkill.Parameter[5].Value := ;
*)



ExecuteSkill();

StepDone := ExecuteSkill.Done;
END_ACTION

ACTION Unblock_active:
StepDone := FALSE;

//Skill auswählen
ExecuteSkill.SkillID 		:= 1316;
ExecuteSkill.SkillName	 	:= 'Unblock';

//Parameter setzen

ExecuteSkill.Parameter[1].ID := 1;
ExecuteSkill.Parameter[1].Name := 'TaskID';
ExecuteSkill.Parameter[1].Value := 125;


(*
ExecuteSkill.Parameter[2].ID := ;
ExecuteSkill.Parameter[2].Name := '';
ExecuteSkill.Parameter[2].Value := ;
*)

(*
ExecuteSkill.Parameter[3].ID := ;
ExecuteSkill.Parameter[3].Name := '';
ExecuteSkill.Parameter[3].Value := ;
*)

(*
ExecuteSkill.Parameter[4].ID := ;
ExecuteSkill.Parameter[4].Name := '';
ExecuteSkill.Parameter[4].Value := ;
*)

(*
ExecuteSkill.Parameter[5].ID := ;
ExecuteSkill.Parameter[5].Name := '';
ExecuteSkill.Parameter[5].Value := ;
*)



ExecuteSkill();

StepDone := ExecuteSkill.Done;
END_ACTION

ACTION Block1_active:
StepDone := FALSE;

//Skill auswählen
ExecuteSkill.SkillID 		:= 1315;
ExecuteSkill.SkillName	 	:= 'Block';

//Parameter setzen

ExecuteSkill.Parameter[1].ID := 1;
ExecuteSkill.Parameter[1].Name := 'TaskID';
ExecuteSkill.Parameter[1].Value := 127;


(*
ExecuteSkill.Parameter[2].ID := ;
ExecuteSkill.Parameter[2].Name := '';
ExecuteSkill.Parameter[2].Value := ;
*)

(*
ExecuteSkill.Parameter[3].ID := ;
ExecuteSkill.Parameter[3].Name := '';
ExecuteSkill.Parameter[3].Value := ;
*)

(*
ExecuteSkill.Parameter[4].ID := ;
ExecuteSkill.Parameter[4].Name := '';
ExecuteSkill.Parameter[4].Value := ;
*)

(*
ExecuteSkill.Parameter[5].ID := ;
ExecuteSkill.Parameter[5].Name := '';
ExecuteSkill.Parameter[5].Value := ;
*)



ExecuteSkill();

StepDone := ExecuteSkill.Done;
END_ACTION

ACTION Block_active:
StepDone := FALSE;

//Skill auswählen
ExecuteSkill.SkillID 		:= 1315;
ExecuteSkill.SkillName	 	:= 'Block';

//Parameter setzen

ExecuteSkill.Parameter[1].ID := 1;
ExecuteSkill.Parameter[1].Name := 'TaskID';
ExecuteSkill.Parameter[1].Value := 124;


(*
ExecuteSkill.Parameter[2].ID := ;
ExecuteSkill.Parameter[2].Name := '';
ExecuteSkill.Parameter[2].Value := ;
*)

(*
ExecuteSkill.Parameter[3].ID := ;
ExecuteSkill.Parameter[3].Name := '';
ExecuteSkill.Parameter[3].Value := ;
*)

(*
ExecuteSkill.Parameter[4].ID := ;
ExecuteSkill.Parameter[4].Name := '';
ExecuteSkill.Parameter[4].Value := ;
*)

(*
ExecuteSkill.Parameter[5].ID := ;
ExecuteSkill.Parameter[5].Name := '';
ExecuteSkill.Parameter[5].Value := ;
*)



ExecuteSkill();

StepDone := ExecuteSkill.Done;
END_ACTION

ACTION Transport2_active:
StepDone := FALSE;

//Skill auswählen
ExecuteSkill.SkillID 		:= 1320;
ExecuteSkill.SkillName	 	:= 'Transport';

//Parameter setzen

ExecuteSkill.Parameter[3].ID := 3;
ExecuteSkill.Parameter[3].Name := 'Velocity';
ExecuteSkill.Parameter[3].Value := 2800;



ExecuteSkill.Parameter[1].ID :=  1;
ExecuteSkill.Parameter[1].Name := 'TargetPosition X';
ExecuteSkill.Parameter[1].Value := 2300 ;



ExecuteSkill.Parameter[2].ID := 2;
ExecuteSkill.Parameter[2].Name := 'TargetPosition Z';
ExecuteSkill.Parameter[2].Value := 0 ;



ExecuteSkill.Parameter[4].ID := 4;
ExecuteSkill.Parameter[4].Name := 'Acceleration';
ExecuteSkill.Parameter[4].Value := 2000 ;


(*
ExecuteSkill.Parameter[5].ID := ;
ExecuteSkill.Parameter[5].Name := '';
ExecuteSkill.Parameter[5].Value := ;
*)



ExecuteSkill();

StepDone := ExecuteSkill.Done;
END_ACTION

ACTION MODULESkill_active:
StepDone := FALSE;
RecipeDone := FALSE;
//Skill auswählen
ExecuteSkill.SkillID 		:= 1337;
ExecuteSkill.SkillName	 	:= 'TESTSKILL1337';

ExecuteSkill();

StepDone := ExecuteSkill.Done;
END_ACTION

END_FUNCTION_BLOCK

// ---- POUs/Recipes/Recipe_10010_transportreserve.TcPOU
FUNCTION_BLOCK Recipe_10010_transportreserve
VAR_INPUT
	execute	: BOOL;
	Order	: DUT_RECIPEORDER;
END_VAR
VAR_OUTPUT
	RecipeInfo	: DUT_RECIPEOFFER;
	RecipeDone	: BOOL;	
	InitDone	: BOOL;
END_VAR
VAR
	StepDone	: BOOL;
END_VAR

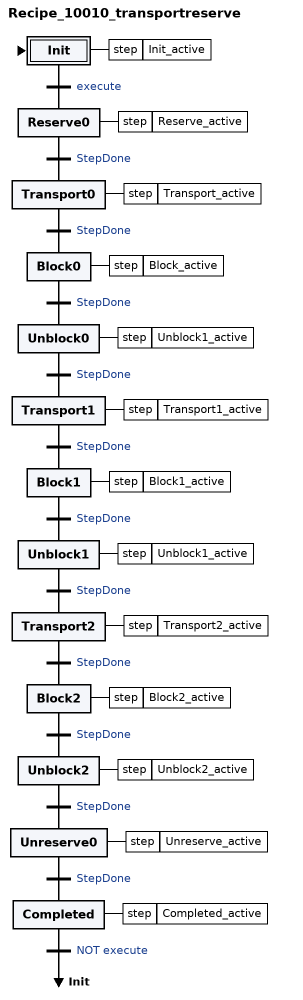
INITIAL_STEP Init:
    Init_active(N);  // step action
END_STEP
TRANSITION FROM Init TO Reserve0
    := execute;
END_TRANSITION
STEP Reserve0:
    Reserve_active(N);  // step action
END_STEP
TRANSITION FROM Reserve0 TO Transport0
    := StepDone;
END_TRANSITION
STEP Transport0:
    Transport_active(N);  // step action
END_STEP
TRANSITION FROM Transport0 TO Block0
    := StepDone;
END_TRANSITION
STEP Block0:
    Block_active(N);  // step action
END_STEP
TRANSITION FROM Block0 TO Unblock0
    := StepDone;
END_TRANSITION
STEP Unblock0:
    Unblock1_active(N);  // step action
END_STEP
TRANSITION FROM Unblock0 TO Transport1
    := StepDone;
END_TRANSITION
STEP Transport1:
    Transport1_active(N);  // step action
END_STEP
TRANSITION FROM Transport1 TO Block1
    := StepDone;
END_TRANSITION
STEP Block1:
    Block1_active(N);  // step action
END_STEP
TRANSITION FROM Block1 TO Unblock1
    := StepDone;
END_TRANSITION
STEP Unblock1:
    Unblock1_active(N);  // step action
END_STEP
TRANSITION FROM Unblock1 TO Transport2
    := StepDone;
END_TRANSITION
STEP Transport2:
    Transport2_active(N);  // step action
END_STEP
TRANSITION FROM Transport2 TO Block2
    := StepDone;
END_TRANSITION
STEP Block2:
    Block2_active(N);  // step action
END_STEP
TRANSITION FROM Block2 TO Unblock2
    := StepDone;
END_TRANSITION
STEP Unblock2:
    Unblock2_active(N);  // step action
END_STEP
TRANSITION FROM Unblock2 TO Unreserve0
    := StepDone;
END_TRANSITION
STEP Unreserve0:
    Unreserve_active(N);  // step action
END_STEP
TRANSITION FROM Unreserve0 TO Completed
    := StepDone;
END_TRANSITION
STEP Completed:
    Completed_active(N);  // step action
END_STEP
TRANSITION FROM Completed TO Init
    := NOT execute;
END_TRANSITION

ACTION Block2_active:
StepDone := FALSE;

//Skill auswählen
ExecuteSkill.SkillID 		:= 1315;
ExecuteSkill.SkillName	 	:= 'Block';

//Parameter setzen

ExecuteSkill.Parameter[1].ID := 1;
ExecuteSkill.Parameter[1].Name := 'TaskID';
ExecuteSkill.Parameter[1].Value := 130;


(*
ExecuteSkill.Parameter[2].ID := ;
ExecuteSkill.Parameter[2].Name := '';
ExecuteSkill.Parameter[2].Value := ;
*)

(*
ExecuteSkill.Parameter[3].ID := ;
ExecuteSkill.Parameter[3].Name := '';
ExecuteSkill.Parameter[3].Value := ;
*)

(*
ExecuteSkill.Parameter[4].ID := ;
ExecuteSkill.Parameter[4].Name := '';
ExecuteSkill.Parameter[4].Value := ;
*)

(*
ExecuteSkill.Parameter[5].ID := ;
ExecuteSkill.Parameter[5].Name := '';
ExecuteSkill.Parameter[5].Value := ;
*)



ExecuteSkill();

StepDone := ExecuteSkill.Done;
END_ACTION

ACTION Unblock_active:
StepDone := FALSE;

//Skill auswählen
ExecuteSkill.SkillID 		:= 1316;
ExecuteSkill.SkillName	 	:= 'Unblock';

//Parameter setzen

ExecuteSkill.Parameter[1].ID := 1;
ExecuteSkill.Parameter[1].Name := 'TaskID';
ExecuteSkill.Parameter[1].Value := 125;


(*
ExecuteSkill.Parameter[2].ID := ;
ExecuteSkill.Parameter[2].Name := '';
ExecuteSkill.Parameter[2].Value := ;
*)

(*
ExecuteSkill.Parameter[3].ID := ;
ExecuteSkill.Parameter[3].Name := '';
ExecuteSkill.Parameter[3].Value := ;
*)

(*
ExecuteSkill.Parameter[4].ID := ;
ExecuteSkill.Parameter[4].Name := '';
ExecuteSkill.Parameter[4].Value := ;
*)

(*
ExecuteSkill.Parameter[5].ID := ;
ExecuteSkill.Parameter[5].Name := '';
ExecuteSkill.Parameter[5].Value := ;
*)



ExecuteSkill();

StepDone := ExecuteSkill.Done;
END_ACTION

ACTION Block_active:
StepDone := FALSE;

//Skill auswählen
ExecuteSkill.SkillID 		:= 1315;
ExecuteSkill.SkillName	 	:= 'Block';

//Parameter setzen

ExecuteSkill.Parameter[1].ID := 1;
ExecuteSkill.Parameter[1].Name := 'TaskID';
ExecuteSkill.Parameter[1].Value := 124;


(*
ExecuteSkill.Parameter[2].ID := ;
ExecuteSkill.Parameter[2].Name := '';
ExecuteSkill.Parameter[2].Value := ;
*)

(*
ExecuteSkill.Parameter[3].ID := ;
ExecuteSkill.Parameter[3].Name := '';
ExecuteSkill.Parameter[3].Value := ;
*)

(*
ExecuteSkill.Parameter[4].ID := ;
ExecuteSkill.Parameter[4].Name := '';
ExecuteSkill.Parameter[4].Value := ;
*)

(*
ExecuteSkill.Parameter[5].ID := ;
ExecuteSkill.Parameter[5].Name := '';
ExecuteSkill.Parameter[5].Value := ;
*)



ExecuteSkill();

StepDone := ExecuteSkill.Done;
END_ACTION

ACTION Transport1_active:
StepDone := FALSE;

//Skill auswählen
ExecuteSkill.SkillID 		:= 1320;
ExecuteSkill.SkillName	 	:= 'Name';

//Parameter setzen

ExecuteSkill.Parameter[3].ID := 3;
ExecuteSkill.Parameter[3].Name := 'Velocity';
ExecuteSkill.Parameter[3].Value := 2500;



ExecuteSkill.Parameter[4].ID := 4 ;
ExecuteSkill.Parameter[4].Name := 'Acceleration';
ExecuteSkill.Parameter[4].Value := 1000 ;



ExecuteSkill.Parameter[1].ID := 1;
ExecuteSkill.Parameter[1].Name := 'TargetPosition X';
ExecuteSkill.Parameter[1].Value := 3200 ;
ExecuteSkill.Parameter[1].StringValue := '#DP#2#XPosition' ;




ExecuteSkill.Parameter[2].ID := 2;
ExecuteSkill.Parameter[2].Name := 'TargetPosition Z';
ExecuteSkill.Parameter[2].Value := 65 ;


(*
ExecuteSkill.Parameter[5].ID := ;
ExecuteSkill.Parameter[5].Name := '';
ExecuteSkill.Parameter[5].Value := ;
*)



ExecuteSkill();

StepDone := ExecuteSkill.Done;
END_ACTION

ACTION Unblock1_active:
StepDone := FALSE;

//Skill auswählen
ExecuteSkill.SkillID 		:= 1316;
ExecuteSkill.SkillName	 	:= 'Unblock';

//Parameter setzen

ExecuteSkill.Parameter[1].ID := 1;
ExecuteSkill.Parameter[1].Name := 'TaskID';
ExecuteSkill.Parameter[1].Value := 128 ;


(*
ExecuteSkill.Parameter[2].ID := ;
ExecuteSkill.Parameter[2].Name := '';
ExecuteSkill.Parameter[2].Value := ;
*)

(*
ExecuteSkill.Parameter[3].ID := ;
ExecuteSkill.Parameter[3].Name := '';
ExecuteSkill.Parameter[3].Value := ;
*)

(*
ExecuteSkill.Parameter[4].ID := ;
ExecuteSkill.Parameter[4].Name := '';
ExecuteSkill.Parameter[4].Value := ;
*)

(*
ExecuteSkill.Parameter[5].ID := ;
ExecuteSkill.Parameter[5].Name := '';
ExecuteSkill.Parameter[5].Value := ;
*)



ExecuteSkill();

StepDone := ExecuteSkill.Done;
END_ACTION

ACTION Transport_active:
StepDone := FALSE;

//Skill auswählen
ExecuteSkill.SkillID 		:= 1320;
ExecuteSkill.SkillName	 	:= 'Transport';

//Parameter setzen
ExecuteSkill.Parameter[3].Dummy := FALSE;
ExecuteSkill.Parameter[3].ID :=3 ;
ExecuteSkill.Parameter[3].Name := 'Velocity';
ExecuteSkill.Parameter[3].Value := 3000;


ExecuteSkill.Parameter[1].Dummy := FALSE;
ExecuteSkill.Parameter[1].ID :=1 ;
ExecuteSkill.Parameter[1].Name := 'TargetPosition X';
ExecuteSkill.Parameter[1].Value := 3300;


ExecuteSkill.Parameter[2].Dummy := FALSE;
ExecuteSkill.Parameter[2].ID := 2 ;
ExecuteSkill.Parameter[2].Name := 'TargetPosition Z';
ExecuteSkill.Parameter[2].Value := 55 ;


ExecuteSkill.Parameter[4].Dummy := FALSE;
ExecuteSkill.Parameter[4].ID := 4 ;
ExecuteSkill.Parameter[4].Name := 'Acceleration';
ExecuteSkill.Parameter[4].Value := 1500;


(*
ExecuteSkill.Parameter[5].ID := ;
ExecuteSkill.Parameter[5].Name := '';
ExecuteSkill.Parameter[5].Value := ;
*)



ExecuteSkill();

StepDone := ExecuteSkill.Done;
END_ACTION

ACTION Unreserve_active:
StepDone := FALSE;

//Skill auswählen
ExecuteSkill.SkillID 		:= 1311;
ExecuteSkill.SkillName	 	:= 'Unreserve';

//Parameter setzen

ExecuteSkill.Parameter[1].ID := 1;
ExecuteSkill.Parameter[1].Name := 'TaskID';
ExecuteSkill.Parameter[1].Value := 131;


(*
ExecuteSkill.Parameter[2].ID := ;
ExecuteSkill.Parameter[2].Name := '';
ExecuteSkill.Parameter[2].Value := ;
*)

(*
ExecuteSkill.Parameter[3].ID := ;
ExecuteSkill.Parameter[3].Name := '';
ExecuteSkill.Parameter[3].Value := ;
*)

(*
ExecuteSkill.Parameter[4].ID := ;
ExecuteSkill.Parameter[4].Name := '';
ExecuteSkill.Parameter[4].Value := ;
*)

(*
ExecuteSkill.Parameter[5].ID := ;
ExecuteSkill.Parameter[5].Name := '';
ExecuteSkill.Parameter[5].Value := ;
*)



ExecuteSkill();

StepDone := ExecuteSkill.Done;
END_ACTION

ACTION MODULESkill_active:
StepDone := FALSE;
RecipeDone := FALSE;
//Skill auswählen
ExecuteSkill.SkillID 		:= 1337;
ExecuteSkill.SkillName	 	:= 'TESTSKILL1337';

ExecuteSkill();

StepDone := ExecuteSkill.Done;
END_ACTION

ACTION Transport2_active:
StepDone := FALSE;

//Skill auswählen
ExecuteSkill.SkillID 		:= 1320;
ExecuteSkill.SkillName	 	:= 'Transport';

//Parameter setzen

ExecuteSkill.Parameter[3].ID := 3;
ExecuteSkill.Parameter[3].Name := 'Velocity';
ExecuteSkill.Parameter[3].Value := 2800;



ExecuteSkill.Parameter[1].ID :=  1;
ExecuteSkill.Parameter[1].Name := 'TargetPosition X';
ExecuteSkill.Parameter[1].Value := 2300 ;



ExecuteSkill.Parameter[2].ID := 2;
ExecuteSkill.Parameter[2].Name := 'TargetPosition Z';
ExecuteSkill.Parameter[2].Value := 0 ;



ExecuteSkill.Parameter[4].ID := 4;
ExecuteSkill.Parameter[4].Name := 'Acceleration';
ExecuteSkill.Parameter[4].Value := 2000 ;


(*
ExecuteSkill.Parameter[5].ID := ;
ExecuteSkill.Parameter[5].Name := '';
ExecuteSkill.Parameter[5].Value := ;
*)



ExecuteSkill();

StepDone := ExecuteSkill.Done;
END_ACTION

ACTION Block1_active:
StepDone := FALSE;

//Skill auswählen
ExecuteSkill.SkillID 		:= 1315;
ExecuteSkill.SkillName	 	:= 'Block';

//Parameter setzen

ExecuteSkill.Parameter[1].ID := 1;
ExecuteSkill.Parameter[1].Name := 'TaskID';
ExecuteSkill.Parameter[1].Value := 127;


(*
ExecuteSkill.Parameter[2].ID := ;
ExecuteSkill.Parameter[2].Name := '';
ExecuteSkill.Parameter[2].Value := ;
*)

(*
ExecuteSkill.Parameter[3].ID := ;
ExecuteSkill.Parameter[3].Name := '';
ExecuteSkill.Parameter[3].Value := ;
*)

(*
ExecuteSkill.Parameter[4].ID := ;
ExecuteSkill.Parameter[4].Name := '';
ExecuteSkill.Parameter[4].Value := ;
*)

(*
ExecuteSkill.Parameter[5].ID := ;
ExecuteSkill.Parameter[5].Name := '';
ExecuteSkill.Parameter[5].Value := ;
*)



ExecuteSkill();

StepDone := ExecuteSkill.Done;
END_ACTION

ACTION Init_active:
RecipeDone := FALSE;

// Initialisation of Recipe Parameters an name etc
RecipeInfo.Name := 'XTS Test Recipe';
RecipeInfo.Description := 'This recipe lets the XTS transport and block/unblock on 3 different stations';
RecipeInfo.Dummy := FALSE;
RecipeInfo.RecipeID := 10010; 	// 
Initdone := TRUE;

//Parameter 1:
(*
	RecipeInfo.UserParameter[1].Dummy 		:= 
	RecipeInfo.UserParameter[1].Default		:=
	RecipeInfo.UserParameter[1].Description	:=
	RecipeInfo.UserParameter[1].MaxValue	:=
	RecipeInfo.UserParameter[1].MinValue	:=
	RecipeInfo.UserParameter[1].Name		:=
	RecipeInfo.UserParameter[1].Unit		:=
*)
//Parameter 2:

(*
	RecipeInfo.UserParameter[2].Dummy 		:= 
	RecipeInfo.UserParameter[2].Default		:=
	RecipeInfo.UserParameter[2].Description	:=
	RecipeInfo.UserParameter[2].MaxValue	:=
	RecipeInfo.UserParameter[2].MinValue	:=
	RecipeInfo.UserParameter[2].Name		:=
	RecipeInfo.UserParameter[2].Unit		:=
*)

//Parameter 3:

(*
	RecipeInfo.UserParameter[3].Dummy 		:= 
	RecipeInfo.UserParameter[3].Default		:=
	RecipeInfo.UserParameter[3].Description	:=
	RecipeInfo.UserParameter[3].MaxValue	:=
	RecipeInfo.UserParameter[3].MinValue	:=
	RecipeInfo.UserParameter[3].Name		:=
	RecipeInfo.UserParameter[3].Unit		:=
*)

//Parameter 4:

(*
	RecipeInfo.UserParameter[4].Dummy 		:= 
	RecipeInfo.UserParameter[4].Default		:=
	RecipeInfo.UserParameter[4].Description	:=
	RecipeInfo.UserParameter[4].MaxValue	:=
	RecipeInfo.UserParameter[4].MinValue	:=
	RecipeInfo.UserParameter[4].Name		:=
	RecipeInfo.UserParameter[4].Unit		:=
*)


//Parameter 5:

(*
	RecipeInfo.UserParameter[5].Dummy 		:= 
	RecipeInfo.UserParameter[5].Default		:=
	RecipeInfo.UserParameter[5].Description	:=
	RecipeInfo.UserParameter[5].MaxValue	:=
	RecipeInfo.UserParameter[5].MinValue	:=
	RecipeInfo.UserParameter[5].Name		:=
	RecipeInfo.UserParameter[5].Unit		:=
*)
END_ACTION

ACTION Unblock2_active:
StepDone := FALSE;

//Skill auswählen
ExecuteSkill.SkillID 		:= 1316;
ExecuteSkill.SkillName	 	:= 'Unblock';

//Parameter setzen

ExecuteSkill.Parameter[1].ID := 1;
ExecuteSkill.Parameter[1].Name := 'TaskID';
ExecuteSkill.Parameter[1].Value := 131;


(*
ExecuteSkill.Parameter[2].ID := ;
ExecuteSkill.Parameter[2].Name := '';
ExecuteSkill.Parameter[2].Value := ;
*)

(*
ExecuteSkill.Parameter[3].ID := ;
ExecuteSkill.Parameter[3].Name := '';
ExecuteSkill.Parameter[3].Value := ;
*)

(*
ExecuteSkill.Parameter[4].ID := ;
ExecuteSkill.Parameter[4].Name := '';
ExecuteSkill.Parameter[4].Value := ;
*)

(*
ExecuteSkill.Parameter[5].ID := ;
ExecuteSkill.Parameter[5].Name := '';
ExecuteSkill.Parameter[5].Value := ;
*)



ExecuteSkill();

StepDone := ExecuteSkill.Done;
END_ACTION

ACTION Completed_active:
RecipeDone := TRUE;
StepDone := FALSE;
END_ACTION

ACTION Reserve_active:
StepDone := FALSE;
RecipeDone := FALSE;
//Skill auswählen
ExecuteSkill.SkillID 		:= 1310;
ExecuteSkill.SkillName	 	:= 'Reserve';

//Parameter setzen

ExecuteSkill.Parameter[1].ID := 1;
ExecuteSkill.Parameter[1].Name := 'TaskID';
ExecuteSkill.Parameter[1].Value := 123;


(*
ExecuteSkill.Parameter[2].ID := ;
ExecuteSkill.Parameter[2].Name := '';
ExecuteSkill.Parameter[2].Value := ;
*)

(*
ExecuteSkill.Parameter[3].ID := ;
ExecuteSkill.Parameter[3].Name := '';
ExecuteSkill.Parameter[3].Value := ;
*)

(*
ExecuteSkill.Parameter[4].ID := ;
ExecuteSkill.Parameter[4].Name := '';
ExecuteSkill.Parameter[4].Value := ;
*)

(*
ExecuteSkill.Parameter[5].ID := ;
ExecuteSkill.Parameter[5].Name := '';
ExecuteSkill.Parameter[5].Value := ;
*)



ExecuteSkill();

StepDone := ExecuteSkill.Done;
END_ACTION

END_FUNCTION_BLOCK

// ---- POUs/Recipes/Recipe_10000_BlankRecipe.TcPOU
FUNCTION_BLOCK Recipe_10000_BlankRecipe
VAR_INPUT
	execute	: BOOL;
	Order	: DUT_RECIPEORDER;
END_VAR
VAR_OUTPUT
	RecipeInfo	: DUT_RECIPEOFFER;
	RecipeDone	: BOOL;	
	InitDone	: BOOL;
END_VAR
VAR
	StepDone	: BOOL;
END_VAR

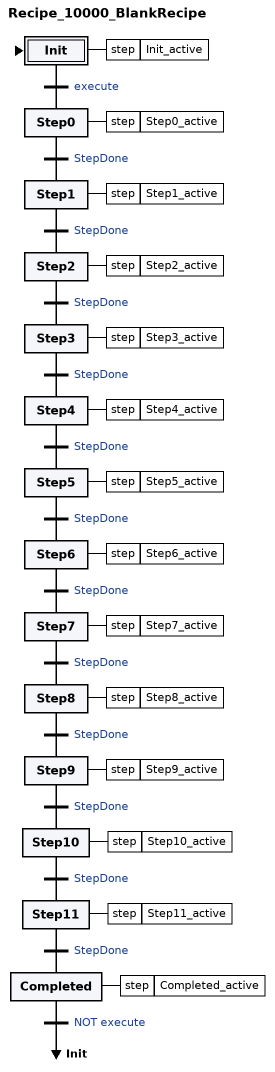
INITIAL_STEP Init:
    Init_active(N);  // step action
END_STEP
TRANSITION FROM Init TO Step0
    := execute;
END_TRANSITION
STEP Step0:
    Step0_active(N);  // step action
END_STEP
TRANSITION FROM Step0 TO Step1
    := StepDone;
END_TRANSITION
STEP Step1:
    Step1_active(N);  // step action
END_STEP
TRANSITION FROM Step1 TO Step2
    := StepDone;
END_TRANSITION
STEP Step2:
    Step2_active(N);  // step action
END_STEP
TRANSITION FROM Step2 TO Step3
    := StepDone;
END_TRANSITION
STEP Step3:
    Step3_active(N);  // step action
END_STEP
TRANSITION FROM Step3 TO Step4
    := StepDone;
END_TRANSITION
STEP Step4:
    Step4_active(N);  // step action
END_STEP
TRANSITION FROM Step4 TO Step5
    := StepDone;
END_TRANSITION
STEP Step5:
    Step5_active(N);  // step action
END_STEP
TRANSITION FROM Step5 TO Step6
    := StepDone;
END_TRANSITION
STEP Step6:
    Step6_active(N);  // step action
END_STEP
TRANSITION FROM Step6 TO Step7
    := StepDone;
END_TRANSITION
STEP Step7:
    Step7_active(N);  // step action
END_STEP
TRANSITION FROM Step7 TO Step8
    := StepDone;
END_TRANSITION
STEP Step8:
    Step8_active(N);  // step action
END_STEP
TRANSITION FROM Step8 TO Step9
    := StepDone;
END_TRANSITION
STEP Step9:
    Step9_active(N);  // step action
END_STEP
TRANSITION FROM Step9 TO Step10
    := StepDone;
END_TRANSITION
STEP Step10:
    Step10_active(N);  // step action
END_STEP
TRANSITION FROM Step10 TO Step11
    := StepDone;
END_TRANSITION
STEP Step11:
    Step11_active(N);  // step action
END_STEP
TRANSITION FROM Step11 TO Completed
    := StepDone;
END_TRANSITION
STEP Completed:
    Completed_active(N);  // step action
END_STEP
TRANSITION FROM Completed TO Init
    := NOT execute;
END_TRANSITION

ACTION Step3_active:
StepDone := FALSE;

//Skill auswählen
ExecuteSkill.SkillID 		:= 0000;
ExecuteSkill.SkillName	 	:= 'Name';

//Parameter setzen
(*
ExecuteSkill.Parameter[1].ID := 3;
ExecuteSkill.Parameter[1].Name := 'Velocity';
ExecuteSkill.Parameter[1].Value := 3000;
*)

(*
ExecuteSkill.Parameter[2].ID := ;
ExecuteSkill.Parameter[2].Name := '';
ExecuteSkill.Parameter[2].Value := ;
*)

(*
ExecuteSkill.Parameter[3].ID := ;
ExecuteSkill.Parameter[3].Name := '';
ExecuteSkill.Parameter[3].Value := ;
*)

(*
ExecuteSkill.Parameter[4].ID := ;
ExecuteSkill.Parameter[4].Name := '';
ExecuteSkill.Parameter[4].Value := ;
*)

(*
ExecuteSkill.Parameter[5].ID := ;
ExecuteSkill.Parameter[5].Name := '';
ExecuteSkill.Parameter[5].Value := ;
*)



ExecuteSkill();

StepDone := ExecuteSkill.Done;
END_ACTION

ACTION Init_active:
RecipeDone := FALSE;

// Initialisation of Recipe Parameters an name etc
RecipeInfo.Name := 'Sample Product Name';
RecipeInfo.Description := 'This Recipe produces a product, which is very productive';
RecipeInfo.Dummy := FALSE;
RecipeInfo.RecipeID := 10000; 	// 
Initdone := TRUE;

//Parameter 1:
(*
	RecipeInfo.UserParameter[1].Dummy 		:= 
	RecipeInfo.UserParameter[1].Default		:=
	RecipeInfo.UserParameter[1].Description	:=
	RecipeInfo.UserParameter[1].MaxValue	:=
	RecipeInfo.UserParameter[1].MinValue	:=
	RecipeInfo.UserParameter[1].Name		:=
	RecipeInfo.UserParameter[1].Unit		:=
*)
//Parameter 2:

(*
	RecipeInfo.UserParameter[2].Dummy 		:= 
	RecipeInfo.UserParameter[2].Default		:=
	RecipeInfo.UserParameter[2].Description	:=
	RecipeInfo.UserParameter[2].MaxValue	:=
	RecipeInfo.UserParameter[2].MinValue	:=
	RecipeInfo.UserParameter[2].Name		:=
	RecipeInfo.UserParameter[2].Unit		:=
*)

//Parameter 3:

(*
	RecipeInfo.UserParameter[3].Dummy 		:= 
	RecipeInfo.UserParameter[3].Default		:=
	RecipeInfo.UserParameter[3].Description	:=
	RecipeInfo.UserParameter[3].MaxValue	:=
	RecipeInfo.UserParameter[3].MinValue	:=
	RecipeInfo.UserParameter[3].Name		:=
	RecipeInfo.UserParameter[3].Unit		:=
*)

//Parameter 4:

(*
	RecipeInfo.UserParameter[4].Dummy 		:= 
	RecipeInfo.UserParameter[4].Default		:=
	RecipeInfo.UserParameter[4].Description	:=
	RecipeInfo.UserParameter[4].MaxValue	:=
	RecipeInfo.UserParameter[4].MinValue	:=
	RecipeInfo.UserParameter[4].Name		:=
	RecipeInfo.UserParameter[4].Unit		:=
*)


//Parameter 5:

(*
	RecipeInfo.UserParameter[5].Dummy 		:= 
	RecipeInfo.UserParameter[5].Default		:=
	RecipeInfo.UserParameter[5].Description	:=
	RecipeInfo.UserParameter[5].MaxValue	:=
	RecipeInfo.UserParameter[5].MinValue	:=
	RecipeInfo.UserParameter[5].Name		:=
	RecipeInfo.UserParameter[5].Unit		:=
*)
END_ACTION

ACTION Step7_active:
StepDone := FALSE;

//Skill auswählen
ExecuteSkill.SkillID 		:= 0000;
ExecuteSkill.SkillName	 	:= 'Name';

//Parameter setzen
(*
ExecuteSkill.Parameter[1].ID := 3;
ExecuteSkill.Parameter[1].Name := 'Velocity';
ExecuteSkill.Parameter[1].Value := 3000;
*)

(*
ExecuteSkill.Parameter[2].ID := ;
ExecuteSkill.Parameter[2].Name := '';
ExecuteSkill.Parameter[2].Value := ;
*)

(*
ExecuteSkill.Parameter[3].ID := ;
ExecuteSkill.Parameter[3].Name := '';
ExecuteSkill.Parameter[3].Value := ;
*)

(*
ExecuteSkill.Parameter[4].ID := ;
ExecuteSkill.Parameter[4].Name := '';
ExecuteSkill.Parameter[4].Value := ;
*)

(*
ExecuteSkill.Parameter[5].ID := ;
ExecuteSkill.Parameter[5].Name := '';
ExecuteSkill.Parameter[5].Value := ;
*)



ExecuteSkill();

StepDone := ExecuteSkill.Done;
END_ACTION

ACTION Step10_active:
StepDone := FALSE;

//Skill auswählen
ExecuteSkill.SkillID 		:= 0000;
ExecuteSkill.SkillName	 	:= 'Name';

//Parameter setzen
(*
ExecuteSkill.Parameter[1].ID := 3;
ExecuteSkill.Parameter[1].Name := 'Velocity';
ExecuteSkill.Parameter[1].Value := 3000;
*)

(*
ExecuteSkill.Parameter[2].ID := ;
ExecuteSkill.Parameter[2].Name := '';
ExecuteSkill.Parameter[2].Value := ;
*)

(*
ExecuteSkill.Parameter[3].ID := ;
ExecuteSkill.Parameter[3].Name := '';
ExecuteSkill.Parameter[3].Value := ;
*)

(*
ExecuteSkill.Parameter[4].ID := ;
ExecuteSkill.Parameter[4].Name := '';
ExecuteSkill.Parameter[4].Value := ;
*)

(*
ExecuteSkill.Parameter[5].ID := ;
ExecuteSkill.Parameter[5].Name := '';
ExecuteSkill.Parameter[5].Value := ;
*)



ExecuteSkill();

StepDone := ExecuteSkill.Done;
END_ACTION

ACTION Step0_active:
StepDone := FALSE;
RecipeDone := FALSE;
//Skill auswählen
ExecuteSkill.SkillID 		:= 0000;
ExecuteSkill.SkillName	 	:= 'Name';

//Parameter setzen
(*
ExecuteSkill.Parameter[1].ID := 3;
ExecuteSkill.Parameter[1].Name := 'Velocity';
ExecuteSkill.Parameter[1].Value := 3000;
*)

(*
ExecuteSkill.Parameter[2].ID := ;
ExecuteSkill.Parameter[2].Name := '';
ExecuteSkill.Parameter[2].Value := ;
*)

(*
ExecuteSkill.Parameter[3].ID := ;
ExecuteSkill.Parameter[3].Name := '';
ExecuteSkill.Parameter[3].Value := ;
*)

(*
ExecuteSkill.Parameter[4].ID := ;
ExecuteSkill.Parameter[4].Name := '';
ExecuteSkill.Parameter[4].Value := ;
*)

(*
ExecuteSkill.Parameter[5].ID := ;
ExecuteSkill.Parameter[5].Name := '';
ExecuteSkill.Parameter[5].Value := ;
*)



ExecuteSkill();

StepDone := ExecuteSkill.Done;
END_ACTION

ACTION Step5_active:
StepDone := FALSE;

//Skill auswählen
ExecuteSkill.SkillID 		:= 0000;
ExecuteSkill.SkillName	 	:= 'Name';

//Parameter setzen
(*
ExecuteSkill.Parameter[1].ID := 3;
ExecuteSkill.Parameter[1].Name := 'Velocity';
ExecuteSkill.Parameter[1].Value := 3000;
*)

(*
ExecuteSkill.Parameter[2].ID := ;
ExecuteSkill.Parameter[2].Name := '';
ExecuteSkill.Parameter[2].Value := ;
*)

(*
ExecuteSkill.Parameter[3].ID := ;
ExecuteSkill.Parameter[3].Name := '';
ExecuteSkill.Parameter[3].Value := ;
*)

(*
ExecuteSkill.Parameter[4].ID := ;
ExecuteSkill.Parameter[4].Name := '';
ExecuteSkill.Parameter[4].Value := ;
*)

(*
ExecuteSkill.Parameter[5].ID := ;
ExecuteSkill.Parameter[5].Name := '';
ExecuteSkill.Parameter[5].Value := ;
*)



ExecuteSkill();

StepDone := ExecuteSkill.Done;
END_ACTION

ACTION Step2_active:
StepDone := FALSE;

//Skill auswählen
ExecuteSkill.SkillID 		:= 0000;
ExecuteSkill.SkillName	 	:= 'Name';

//Parameter setzen
(*
ExecuteSkill.Parameter[1].ID := 3;
ExecuteSkill.Parameter[1].Name := 'Velocity';
ExecuteSkill.Parameter[1].Value := 3000;
*)

(*
ExecuteSkill.Parameter[2].ID := ;
ExecuteSkill.Parameter[2].Name := '';
ExecuteSkill.Parameter[2].Value := ;
*)

(*
ExecuteSkill.Parameter[3].ID := ;
ExecuteSkill.Parameter[3].Name := '';
ExecuteSkill.Parameter[3].Value := ;
*)

(*
ExecuteSkill.Parameter[4].ID := ;
ExecuteSkill.Parameter[4].Name := '';
ExecuteSkill.Parameter[4].Value := ;
*)

(*
ExecuteSkill.Parameter[5].ID := ;
ExecuteSkill.Parameter[5].Name := '';
ExecuteSkill.Parameter[5].Value := ;
*)



ExecuteSkill();

StepDone := ExecuteSkill.Done;
END_ACTION

ACTION Step4_active:
StepDone := FALSE;

//Skill auswählen
ExecuteSkill.SkillID 		:= 0000;
ExecuteSkill.SkillName	 	:= 'Name';

//Parameter setzen
(*
ExecuteSkill.Parameter[1].ID := 3;
ExecuteSkill.Parameter[1].Name := 'Velocity';
ExecuteSkill.Parameter[1].Value := 3000;
*)

(*
ExecuteSkill.Parameter[2].ID := ;
ExecuteSkill.Parameter[2].Name := '';
ExecuteSkill.Parameter[2].Value := ;
*)

(*
ExecuteSkill.Parameter[3].ID := ;
ExecuteSkill.Parameter[3].Name := '';
ExecuteSkill.Parameter[3].Value := ;
*)

(*
ExecuteSkill.Parameter[4].ID := ;
ExecuteSkill.Parameter[4].Name := '';
ExecuteSkill.Parameter[4].Value := ;
*)

(*
ExecuteSkill.Parameter[5].ID := ;
ExecuteSkill.Parameter[5].Name := '';
ExecuteSkill.Parameter[5].Value := ;
*)



ExecuteSkill();

StepDone := ExecuteSkill.Done;
END_ACTION

ACTION Step8_active:
StepDone := FALSE;

//Skill auswählen
ExecuteSkill.SkillID 		:= 0000;
ExecuteSkill.SkillName	 	:= 'Name';

//Parameter setzen
(*
ExecuteSkill.Parameter[1].ID := 3;
ExecuteSkill.Parameter[1].Name := 'Velocity';
ExecuteSkill.Parameter[1].Value := 3000;
*)

(*
ExecuteSkill.Parameter[2].ID := ;
ExecuteSkill.Parameter[2].Name := '';
ExecuteSkill.Parameter[2].Value := ;
*)

(*
ExecuteSkill.Parameter[3].ID := ;
ExecuteSkill.Parameter[3].Name := '';
ExecuteSkill.Parameter[3].Value := ;
*)

(*
ExecuteSkill.Parameter[4].ID := ;
ExecuteSkill.Parameter[4].Name := '';
ExecuteSkill.Parameter[4].Value := ;
*)

(*
ExecuteSkill.Parameter[5].ID := ;
ExecuteSkill.Parameter[5].Name := '';
ExecuteSkill.Parameter[5].Value := ;
*)



ExecuteSkill();

StepDone := ExecuteSkill.Done;
END_ACTION

ACTION Step1_active:
StepDone := FALSE;

//Skill auswählen
ExecuteSkill.SkillID 		:= 0000;
ExecuteSkill.SkillName	 	:= 'Name';

//Parameter setzen
(*
ExecuteSkill.Parameter[1].ID := 3;
ExecuteSkill.Parameter[1].Name := 'Velocity';
ExecuteSkill.Parameter[1].Value := 3000;
*)

(*
ExecuteSkill.Parameter[2].ID := ;
ExecuteSkill.Parameter[2].Name := '';
ExecuteSkill.Parameter[2].Value := ;
*)

(*
ExecuteSkill.Parameter[3].ID := ;
ExecuteSkill.Parameter[3].Name := '';
ExecuteSkill.Parameter[3].Value := ;
*)

(*
ExecuteSkill.Parameter[4].ID := ;
ExecuteSkill.Parameter[4].Name := '';
ExecuteSkill.Parameter[4].Value := ;
*)

(*
ExecuteSkill.Parameter[5].ID := ;
ExecuteSkill.Parameter[5].Name := '';
ExecuteSkill.Parameter[5].Value := ;
*)



ExecuteSkill();

StepDone := ExecuteSkill.Done;
END_ACTION

ACTION Step11_active:
StepDone := FALSE;

//Skill auswählen
ExecuteSkill.SkillID 		:= 0000;
ExecuteSkill.SkillName	 	:= 'Name';

//Parameter setzen
(*
ExecuteSkill.Parameter[1].ID := 3;
ExecuteSkill.Parameter[1].Name := 'Velocity';
ExecuteSkill.Parameter[1].Value := 3000;
*)

(*
ExecuteSkill.Parameter[2].ID := ;
ExecuteSkill.Parameter[2].Name := '';
ExecuteSkill.Parameter[2].Value := ;
*)

(*
ExecuteSkill.Parameter[3].ID := ;
ExecuteSkill.Parameter[3].Name := '';
ExecuteSkill.Parameter[3].Value := ;
*)

(*
ExecuteSkill.Parameter[4].ID := ;
ExecuteSkill.Parameter[4].Name := '';
ExecuteSkill.Parameter[4].Value := ;
*)

(*
ExecuteSkill.Parameter[5].ID := ;
ExecuteSkill.Parameter[5].Name := '';
ExecuteSkill.Parameter[5].Value := ;
*)



ExecuteSkill();

StepDone := ExecuteSkill.Done;
END_ACTION

ACTION Completed_active:
RecipeDone := TRUE;
StepDone := FALSE;
END_ACTION

ACTION Step9_active:
StepDone := FALSE;

//Skill auswählen
ExecuteSkill.SkillID 		:= 0000;
ExecuteSkill.SkillName	 	:= 'Name';

//Parameter setzen
(*
ExecuteSkill.Parameter[1].ID := 3;
ExecuteSkill.Parameter[1].Name := 'Velocity';
ExecuteSkill.Parameter[1].Value := 3000;
*)

(*
ExecuteSkill.Parameter[2].ID := ;
ExecuteSkill.Parameter[2].Name := '';
ExecuteSkill.Parameter[2].Value := ;
*)

(*
ExecuteSkill.Parameter[3].ID := ;
ExecuteSkill.Parameter[3].Name := '';
ExecuteSkill.Parameter[3].Value := ;
*)

(*
ExecuteSkill.Parameter[4].ID := ;
ExecuteSkill.Parameter[4].Name := '';
ExecuteSkill.Parameter[4].Value := ;
*)

(*
ExecuteSkill.Parameter[5].ID := ;
ExecuteSkill.Parameter[5].Name := '';
ExecuteSkill.Parameter[5].Value := ;
*)



ExecuteSkill();

StepDone := ExecuteSkill.Done;
END_ACTION

ACTION Step6_active:
StepDone := FALSE;

//Skill auswählen
ExecuteSkill.SkillID 		:= 0000;
ExecuteSkill.SkillName	 	:= 'Name';

//Parameter setzen
(*
ExecuteSkill.Parameter[1].ID := 3;
ExecuteSkill.Parameter[1].Name := 'Velocity';
ExecuteSkill.Parameter[1].Value := 3000;
*)

(*
ExecuteSkill.Parameter[2].ID := ;
ExecuteSkill.Parameter[2].Name := '';
ExecuteSkill.Parameter[2].Value := ;
*)

(*
ExecuteSkill.Parameter[3].ID := ;
ExecuteSkill.Parameter[3].Name := '';
ExecuteSkill.Parameter[3].Value := ;
*)

(*
ExecuteSkill.Parameter[4].ID := ;
ExecuteSkill.Parameter[4].Name := '';
ExecuteSkill.Parameter[4].Value := ;
*)

(*
ExecuteSkill.Parameter[5].ID := ;
ExecuteSkill.Parameter[5].Name := '';
ExecuteSkill.Parameter[5].Value := ;
*)



ExecuteSkill();

StepDone := ExecuteSkill.Done;
END_ACTION

END_FUNCTION_BLOCK

// ---- POUs/Recipes/Recipe_10011_Skill1337.TcPOU
FUNCTION_BLOCK Recipe_10011_Skill1337
VAR_INPUT
	execute	: BOOL;
	Order	: DUT_RECIPEORDER;
END_VAR
VAR_OUTPUT
	RecipeInfo	: DUT_RECIPEOFFER;
	RecipeDone	: BOOL;	
	InitDone	: BOOL;
END_VAR
VAR
	StepDone	: BOOL;
END_VAR

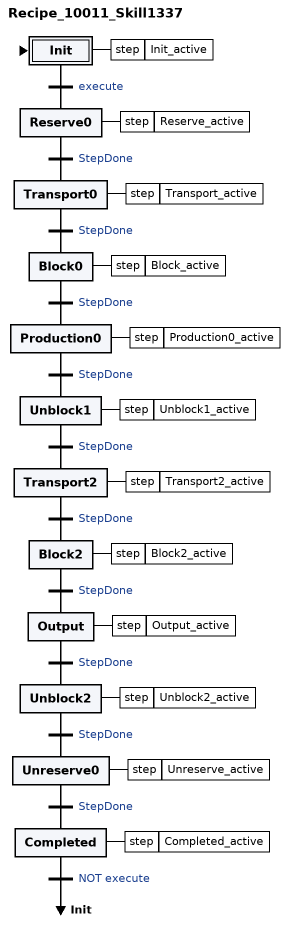
INITIAL_STEP Init:
    Init_active(N);  // step action
END_STEP
TRANSITION FROM Init TO Reserve0
    := execute;
END_TRANSITION
STEP Reserve0:
    Reserve_active(N);  // step action
END_STEP
TRANSITION FROM Reserve0 TO Transport0
    := StepDone;
END_TRANSITION
STEP Transport0:
    Transport_active(N);  // step action
END_STEP
TRANSITION FROM Transport0 TO Block0
    := StepDone;
END_TRANSITION
STEP Block0:
    Block_active(N);  // step action
END_STEP
TRANSITION FROM Block0 TO Production0
    := StepDone;
END_TRANSITION
STEP Production0:
    Production0_active(N);  // step action
END_STEP
TRANSITION FROM Production0 TO Unblock1
    := StepDone;
END_TRANSITION
STEP Unblock1:
    Unblock1_active(N);  // step action
END_STEP
TRANSITION FROM Unblock1 TO Transport2
    := StepDone;
END_TRANSITION
STEP Transport2:
    Transport2_active(N);  // step action
END_STEP
TRANSITION FROM Transport2 TO Block2
    := StepDone;
END_TRANSITION
STEP Block2:
    Block2_active(N);  // step action
END_STEP
TRANSITION FROM Block2 TO Output
    := StepDone;
END_TRANSITION
STEP Output:
    Output_active(N);  // step action
END_STEP
TRANSITION FROM Output TO Unblock2
    := StepDone;
END_TRANSITION
STEP Unblock2:
    Unblock2_active(N);  // step action
END_STEP
TRANSITION FROM Unblock2 TO Unreserve0
    := StepDone;
END_TRANSITION
STEP Unreserve0:
    Unreserve_active(N);  // step action
END_STEP
TRANSITION FROM Unreserve0 TO Completed
    := StepDone;
END_TRANSITION
STEP Completed:
    Completed_active(N);  // step action
END_STEP
TRANSITION FROM Completed TO Init
    := NOT execute;
END_TRANSITION

ACTION Transport_active:
StepDone := FALSE;

//Skill auswählen
ExecuteSkill.SkillID 		:= 1320;
ExecuteSkill.SkillName	 	:= 'Transport';

//Parameter setzen

ExecuteSkill.Parameter[3].ID :=3 ;
ExecuteSkill.Parameter[3].Name := 'Velocity';
ExecuteSkill.Parameter[3].Value := 3000;



ExecuteSkill.Parameter[1].ID :=1 ;
ExecuteSkill.Parameter[1].Name := 'TargetPosition X';
ExecuteSkill.Parameter[1].Value := 2000;
ExecuteSkill.Parameter[1].StringValue := '#DP#2#XPosition';



ExecuteSkill.Parameter[2].ID := 2 ;
ExecuteSkill.Parameter[2].Name := 'TargetPosition Z';
ExecuteSkill.Parameter[2].Value := 0 ;



ExecuteSkill.Parameter[4].ID := 4 ;
ExecuteSkill.Parameter[4].Name := 'Acceleration';
ExecuteSkill.Parameter[4].Value := 1500;


(*
ExecuteSkill.Parameter[5].ID := ;
ExecuteSkill.Parameter[5].Name := '';
ExecuteSkill.Parameter[5].Value := ;
*)



ExecuteSkill();

StepDone := ExecuteSkill.Done;
END_ACTION

ACTION Transport1_active:
StepDone := FALSE;

//Skill auswählen
ExecuteSkill.SkillID 		:= 1320;
ExecuteSkill.SkillName	 	:= 'Name';

//Parameter setzen

ExecuteSkill.Parameter[3].ID := 3;
ExecuteSkill.Parameter[3].Name := 'Velocity';
ExecuteSkill.Parameter[3].Value := 2500;



ExecuteSkill.Parameter[4].ID := 4 ;
ExecuteSkill.Parameter[4].Name := 'Acceleration';
ExecuteSkill.Parameter[4].Value := 1000 ;



ExecuteSkill.Parameter[1].ID := 1;
ExecuteSkill.Parameter[1].Name := 'TargetPosition X';
ExecuteSkill.Parameter[1].Value := 3200 ;
ExecuteSkill.Parameter[1].StringValue := '#DP#2#XPosition' ;




ExecuteSkill.Parameter[2].ID := 2;
ExecuteSkill.Parameter[2].Name := 'TargetPosition Z';
ExecuteSkill.Parameter[2].Value := 65 ;


(*
ExecuteSkill.Parameter[5].ID := ;
ExecuteSkill.Parameter[5].Name := '';
ExecuteSkill.Parameter[5].Value := ;
*)



ExecuteSkill();

StepDone := ExecuteSkill.Done;
END_ACTION

ACTION Block2_active:
StepDone := FALSE;

//Skill auswählen
ExecuteSkill.SkillID 		:= 1315;
ExecuteSkill.SkillName	 	:= 'Block';

//Parameter setzen

ExecuteSkill.Parameter[1].ID := 1;
ExecuteSkill.Parameter[1].Name := 'TaskID';
ExecuteSkill.Parameter[1].Value := 130;


(*
ExecuteSkill.Parameter[2].ID := ;
ExecuteSkill.Parameter[2].Name := '';
ExecuteSkill.Parameter[2].Value := ;
*)

(*
ExecuteSkill.Parameter[3].ID := ;
ExecuteSkill.Parameter[3].Name := '';
ExecuteSkill.Parameter[3].Value := ;
*)

(*
ExecuteSkill.Parameter[4].ID := ;
ExecuteSkill.Parameter[4].Name := '';
ExecuteSkill.Parameter[4].Value := ;
*)

(*
ExecuteSkill.Parameter[5].ID := ;
ExecuteSkill.Parameter[5].Name := '';
ExecuteSkill.Parameter[5].Value := ;
*)



ExecuteSkill();

StepDone := ExecuteSkill.Done;
END_ACTION

ACTION Unblock1_active:
StepDone := FALSE;

//Skill auswählen
ExecuteSkill.SkillID 		:= 1316;
ExecuteSkill.SkillName	 	:= 'Unblock';

//Parameter setzen

ExecuteSkill.Parameter[1].ID := 1;
ExecuteSkill.Parameter[1].Name := 'TaskID';
ExecuteSkill.Parameter[1].Value := 128 ;


(*
ExecuteSkill.Parameter[2].ID := ;
ExecuteSkill.Parameter[2].Name := '';
ExecuteSkill.Parameter[2].Value := ;
*)

(*
ExecuteSkill.Parameter[3].ID := ;
ExecuteSkill.Parameter[3].Name := '';
ExecuteSkill.Parameter[3].Value := ;
*)

(*
ExecuteSkill.Parameter[4].ID := ;
ExecuteSkill.Parameter[4].Name := '';
ExecuteSkill.Parameter[4].Value := ;
*)

(*
ExecuteSkill.Parameter[5].ID := ;
ExecuteSkill.Parameter[5].Name := '';
ExecuteSkill.Parameter[5].Value := ;
*)



ExecuteSkill();

StepDone := ExecuteSkill.Done;
END_ACTION

ACTION Reserve_active:
StepDone := FALSE;
RecipeDone := FALSE;
//Skill auswählen
ExecuteSkill.SkillID 		:= 1310;
ExecuteSkill.SkillName	 	:= 'Reserve';

//Parameter setzen

ExecuteSkill.Parameter[1].ID := 1;
ExecuteSkill.Parameter[1].Name := 'TaskID';
ExecuteSkill.Parameter[1].Value := 123;


(*
ExecuteSkill.Parameter[2].ID := ;
ExecuteSkill.Parameter[2].Name := '';
ExecuteSkill.Parameter[2].Value := ;
*)

(*
ExecuteSkill.Parameter[3].ID := ;
ExecuteSkill.Parameter[3].Name := '';
ExecuteSkill.Parameter[3].Value := ;
*)

(*
ExecuteSkill.Parameter[4].ID := ;
ExecuteSkill.Parameter[4].Name := '';
ExecuteSkill.Parameter[4].Value := ;
*)

(*
ExecuteSkill.Parameter[5].ID := ;
ExecuteSkill.Parameter[5].Name := '';
ExecuteSkill.Parameter[5].Value := ;
*)



ExecuteSkill();

StepDone := ExecuteSkill.Done;
END_ACTION

ACTION Output_active:
StepDone := FALSE;

//Skill auswählen
ExecuteSkill.SkillID 		:= 1403;
ExecuteSkill.SkillName	 	:= 'Output';

//Parameter setzen

ExecuteSkill.Parameter[1].ID := 1;
ExecuteSkill.Parameter[1].Name := 'TaskID';
ExecuteSkill.Parameter[1].Value := Order.TaskID;




ExecuteSkill();

StepDone := ExecuteSkill.Done;
END_ACTION

ACTION Unreserve_active:
StepDone := FALSE;

//Skill auswählen
ExecuteSkill.SkillID 		:= 1311;
ExecuteSkill.SkillName	 	:= 'Unreserve';

//Parameter setzen

ExecuteSkill.Parameter[1].ID := 1;
ExecuteSkill.Parameter[1].Name := 'TaskID';
ExecuteSkill.Parameter[1].Value := 131;


(*
ExecuteSkill.Parameter[2].ID := ;
ExecuteSkill.Parameter[2].Name := '';
ExecuteSkill.Parameter[2].Value := ;
*)

(*
ExecuteSkill.Parameter[3].ID := ;
ExecuteSkill.Parameter[3].Name := '';
ExecuteSkill.Parameter[3].Value := ;
*)

(*
ExecuteSkill.Parameter[4].ID := ;
ExecuteSkill.Parameter[4].Name := '';
ExecuteSkill.Parameter[4].Value := ;
*)

(*
ExecuteSkill.Parameter[5].ID := ;
ExecuteSkill.Parameter[5].Name := '';
ExecuteSkill.Parameter[5].Value := ;
*)



ExecuteSkill();

StepDone := ExecuteSkill.Done;
END_ACTION

ACTION Block_active:
StepDone := FALSE;

//Skill auswählen
ExecuteSkill.SkillID 		:= 1315;
ExecuteSkill.SkillName	 	:= 'Block';

//Parameter setzen

ExecuteSkill.Parameter[1].ID := 1;
ExecuteSkill.Parameter[1].Name := 'TaskID';
ExecuteSkill.Parameter[1].Value := 124;


(*
ExecuteSkill.Parameter[2].ID := ;
ExecuteSkill.Parameter[2].Name := '';
ExecuteSkill.Parameter[2].Value := ;
*)

(*
ExecuteSkill.Parameter[3].ID := ;
ExecuteSkill.Parameter[3].Name := '';
ExecuteSkill.Parameter[3].Value := ;
*)

(*
ExecuteSkill.Parameter[4].ID := ;
ExecuteSkill.Parameter[4].Name := '';
ExecuteSkill.Parameter[4].Value := ;
*)

(*
ExecuteSkill.Parameter[5].ID := ;
ExecuteSkill.Parameter[5].Name := '';
ExecuteSkill.Parameter[5].Value := ;
*)



ExecuteSkill();

StepDone := ExecuteSkill.Done;
END_ACTION

ACTION Meinskill_active:
StepDone := FALSE;
RecipeDone := FALSE;
//Skill auswählen
ExecuteSkill.SkillID 		:= 1337;
ExecuteSkill.SkillName	 	:= 'ParameterTESTSKILL1337';


ExecuteSkill.Parameter[0].ID := 10;
ExecuteSkill.Parameter[0].Name := 'Blinkfrequenz';
ExecuteSkill.Parameter[0].Value := Order.UserParameter[0].Value;


ExecuteSkill();

StepDone := ExecuteSkill.Done;
END_ACTION

ACTION Unblock_active:
StepDone := FALSE;

//Skill auswählen
ExecuteSkill.SkillID 		:= 1316;
ExecuteSkill.SkillName	 	:= 'Unblock';

//Parameter setzen

ExecuteSkill.Parameter[1].ID := 1;
ExecuteSkill.Parameter[1].Name := 'TaskID';
ExecuteSkill.Parameter[1].Value := 125;


(*
ExecuteSkill.Parameter[2].ID := ;
ExecuteSkill.Parameter[2].Name := '';
ExecuteSkill.Parameter[2].Value := ;
*)

(*
ExecuteSkill.Parameter[3].ID := ;
ExecuteSkill.Parameter[3].Name := '';
ExecuteSkill.Parameter[3].Value := ;
*)

(*
ExecuteSkill.Parameter[4].ID := ;
ExecuteSkill.Parameter[4].Name := '';
ExecuteSkill.Parameter[4].Value := ;
*)

(*
ExecuteSkill.Parameter[5].ID := ;
ExecuteSkill.Parameter[5].Name := '';
ExecuteSkill.Parameter[5].Value := ;
*)



ExecuteSkill();

StepDone := ExecuteSkill.Done;
END_ACTION

ACTION Unblock2_active:
StepDone := FALSE;

//Skill auswählen
ExecuteSkill.SkillID 		:= 1316;
ExecuteSkill.SkillName	 	:= 'Unblock';

//Parameter setzen

ExecuteSkill.Parameter[1].ID := 1;
ExecuteSkill.Parameter[1].Name := 'TaskID';
ExecuteSkill.Parameter[1].Value := 131;


(*
ExecuteSkill.Parameter[2].ID := ;
ExecuteSkill.Parameter[2].Name := '';
ExecuteSkill.Parameter[2].Value := ;
*)

(*
ExecuteSkill.Parameter[3].ID := ;
ExecuteSkill.Parameter[3].Name := '';
ExecuteSkill.Parameter[3].Value := ;
*)

(*
ExecuteSkill.Parameter[4].ID := ;
ExecuteSkill.Parameter[4].Name := '';
ExecuteSkill.Parameter[4].Value := ;
*)

(*
ExecuteSkill.Parameter[5].ID := ;
ExecuteSkill.Parameter[5].Name := '';
ExecuteSkill.Parameter[5].Value := ;
*)



ExecuteSkill();

StepDone := ExecuteSkill.Done;
END_ACTION

ACTION Init_active:
RecipeDone := FALSE;

// Initialisation of Recipe Parameters an name etc
RecipeInfo.Name := 'Simulation module x Test recipe';
RecipeInfo.Description := 'Execution of  skill 1337 for Simulation Testing';
RecipeInfo.Dummy := FALSE;
RecipeInfo.RecipeID := 10011; 	// 
Initdone := TRUE;

//Parameter 0:

	RecipeInfo.UserParameter[0].Dummy 		:= FALSE;
	RecipeInfo.UserParameter[0].Default		:= 0.5;
	RecipeInfo.UserParameter[0].Description	:= 'Simulation blinking frequency';
	RecipeInfo.UserParameter[0].MaxValue	:= 50.0;
	RecipeInfo.UserParameter[0].MinValue	:= 0;
	RecipeInfo.UserParameter[0].Name		:= 'Production Frequenz';
	RecipeInfo.UserParameter[0].Unit		:= 'HZ';
	RecipeInfo.UserParameter[0].Step		:= 1;

//Parameter 1:
(*
	RecipeInfo.UserParameter[1].Dummy 		:= 
	RecipeInfo.UserParameter[1].Default		:=
	RecipeInfo.UserParameter[1].Description	:=
	RecipeInfo.UserParameter[1].MaxValue	:=
	RecipeInfo.UserParameter[1].MinValue	:=
	RecipeInfo.UserParameter[1].Name		:=
	RecipeInfo.UserParameter[1].Unit		:=
*)
	

//Parameter 2:

(*
	RecipeInfo.UserParameter[2].Dummy 		:= 
	RecipeInfo.UserParameter[2].Default		:=
	RecipeInfo.UserParameter[2].Description	:=
	RecipeInfo.UserParameter[2].MaxValue	:=
	RecipeInfo.UserParameter[2].MinValue	:=
	RecipeInfo.UserParameter[2].Name		:=
	RecipeInfo.UserParameter[2].Unit		:=
*)

//Parameter 3:

(*
	RecipeInfo.UserParameter[3].Dummy 		:= 
	RecipeInfo.UserParameter[3].Default		:=
	RecipeInfo.UserParameter[3].Description	:=
	RecipeInfo.UserParameter[3].MaxValue	:=
	RecipeInfo.UserParameter[3].MinValue	:=
	RecipeInfo.UserParameter[3].Name		:=
	RecipeInfo.UserParameter[3].Unit		:=
*)

//Parameter 4:

(*
	RecipeInfo.UserParameter[4].Dummy 		:= 
	RecipeInfo.UserParameter[4].Default		:=
	RecipeInfo.UserParameter[4].Description	:=
	RecipeInfo.UserParameter[4].MaxValue	:=
	RecipeInfo.UserParameter[4].MinValue	:=
	RecipeInfo.UserParameter[4].Name		:=
	RecipeInfo.UserParameter[4].Unit		:=
*)


//Parameter 5:

(*
	RecipeInfo.UserParameter[5].Dummy 		:= 
	RecipeInfo.UserParameter[5].Default		:=
	RecipeInfo.UserParameter[5].Description	:=
	RecipeInfo.UserParameter[5].MaxValue	:=
	RecipeInfo.UserParameter[5].MinValue	:=
	RecipeInfo.UserParameter[5].Name		:=
	RecipeInfo.UserParameter[5].Unit		:=
*)
END_ACTION

ACTION Completed_active:
RecipeDone := TRUE;
StepDone := FALSE;
END_ACTION

ACTION Production0_active:
StepDone := FALSE;
RecipeDone := FALSE;
//Skill auswählen
ExecuteSkill.SkillID 		:= 1337;
ExecuteSkill.SkillName	 	:= 'ParameterTESTSKILL1337';


ExecuteSkill.Parameter[0].ID := 10;
ExecuteSkill.Parameter[0].Name := 'Blinkfrequenz';
ExecuteSkill.Parameter[0].Value := Order.UserParameter[0].Value;


ExecuteSkill();

StepDone := ExecuteSkill.Done;
END_ACTION

ACTION Block1_active:
StepDone := FALSE;

//Skill auswählen
ExecuteSkill.SkillID 		:= 1315;
ExecuteSkill.SkillName	 	:= 'Block';

//Parameter setzen

ExecuteSkill.Parameter[1].ID := 1;
ExecuteSkill.Parameter[1].Name := 'TaskID';
ExecuteSkill.Parameter[1].Value := 127;


(*
ExecuteSkill.Parameter[2].ID := ;
ExecuteSkill.Parameter[2].Name := '';
ExecuteSkill.Parameter[2].Value := ;
*)

(*
ExecuteSkill.Parameter[3].ID := ;
ExecuteSkill.Parameter[3].Name := '';
ExecuteSkill.Parameter[3].Value := ;
*)

(*
ExecuteSkill.Parameter[4].ID := ;
ExecuteSkill.Parameter[4].Name := '';
ExecuteSkill.Parameter[4].Value := ;
*)

(*
ExecuteSkill.Parameter[5].ID := ;
ExecuteSkill.Parameter[5].Name := '';
ExecuteSkill.Parameter[5].Value := ;
*)



ExecuteSkill();

StepDone := ExecuteSkill.Done;
END_ACTION

ACTION Transport2_active:
StepDone := FALSE;

//Skill auswählen
ExecuteSkill.SkillID 		:= 1320;
ExecuteSkill.SkillName	 	:= 'Transport';

//Parameter setzen

ExecuteSkill.Parameter[3].ID := 3;
ExecuteSkill.Parameter[3].Name := 'Velocity';
ExecuteSkill.Parameter[3].Value := 2800;



ExecuteSkill.Parameter[1].ID :=  1;
ExecuteSkill.Parameter[1].Name := 'TargetPosition X';
ExecuteSkill.Parameter[1].Value := 30 ;
ExecuteSkill.Parameter[1].StringValue := '#DP#2#XPosition';



ExecuteSkill.Parameter[2].ID := 2;
ExecuteSkill.Parameter[2].Name := 'TargetPosition Z';
ExecuteSkill.Parameter[2].Value := ZInputOutput;



ExecuteSkill.Parameter[4].ID := 4;
ExecuteSkill.Parameter[4].Name := 'Acceleration';
ExecuteSkill.Parameter[4].Value := 2000 ;


(*
ExecuteSkill.Parameter[5].ID := ;
ExecuteSkill.Parameter[5].Name := '';
ExecuteSkill.Parameter[5].Value := ;
*)



ExecuteSkill();

StepDone := ExecuteSkill.Done;
END_ACTION

END_FUNCTION_BLOCK

// ---- POUs/Testing.TcPOU
PROGRAM Testing
VAR
	
	StartTestSequence: BOOL;
	IterationCount	: UINT;
	RecipeID		: INT := 10001;
	
	NoOPC			: BOOL;
	state		: INT;
	OrderCnt	: UINT := 9000;
	
	TempCounter	: UINT;
END_VAR

CASE state OF
	

	0: 
		IF StartTestSequence AND NoOPC THEN
			state := 1;
		END_IF
		
	1:	
		IF Tempcounter < IterationCount THEN
			IF NOT Queue.Pending THEN
				Queue.Pending 	:= TRUE;
				Queue.RecipeID 	:= RecipeID;
				Queue.TaskID 	:= OrderCnt;
				Queue.Name		:= 'Testorder';
				Tempcounter 	:= TempCounter +1;
				OrderCnt 		:= OrderCnt +1;
				
			END_IF
		ELSE
			TempCounter 		:= 0;
			state 				:= 0;
			StartTestSequence 	:= FALSE;
		END_IF
		
		
	
	
END_CASE

END_PROGRAM

// ---- POUs/Recipes/Recipe_10017_DoubleCookiemitTopping.TcPOU
FUNCTION_BLOCK Recipe_10017_DoubleCookiemitTopping
VAR_INPUT
	execute	: BOOL;
	Order	: DUT_RECIPEORDER;
END_VAR
VAR_OUTPUT
	RecipeInfo	: DUT_RECIPEOFFER;
	RecipeDone	: BOOL;	
	InitDone	: BOOL;
END_VAR
VAR
	StepDone	: BOOL;
	Layercnt	: INT := 0;
	OrderLayers	: INT := 1;
END_VAR

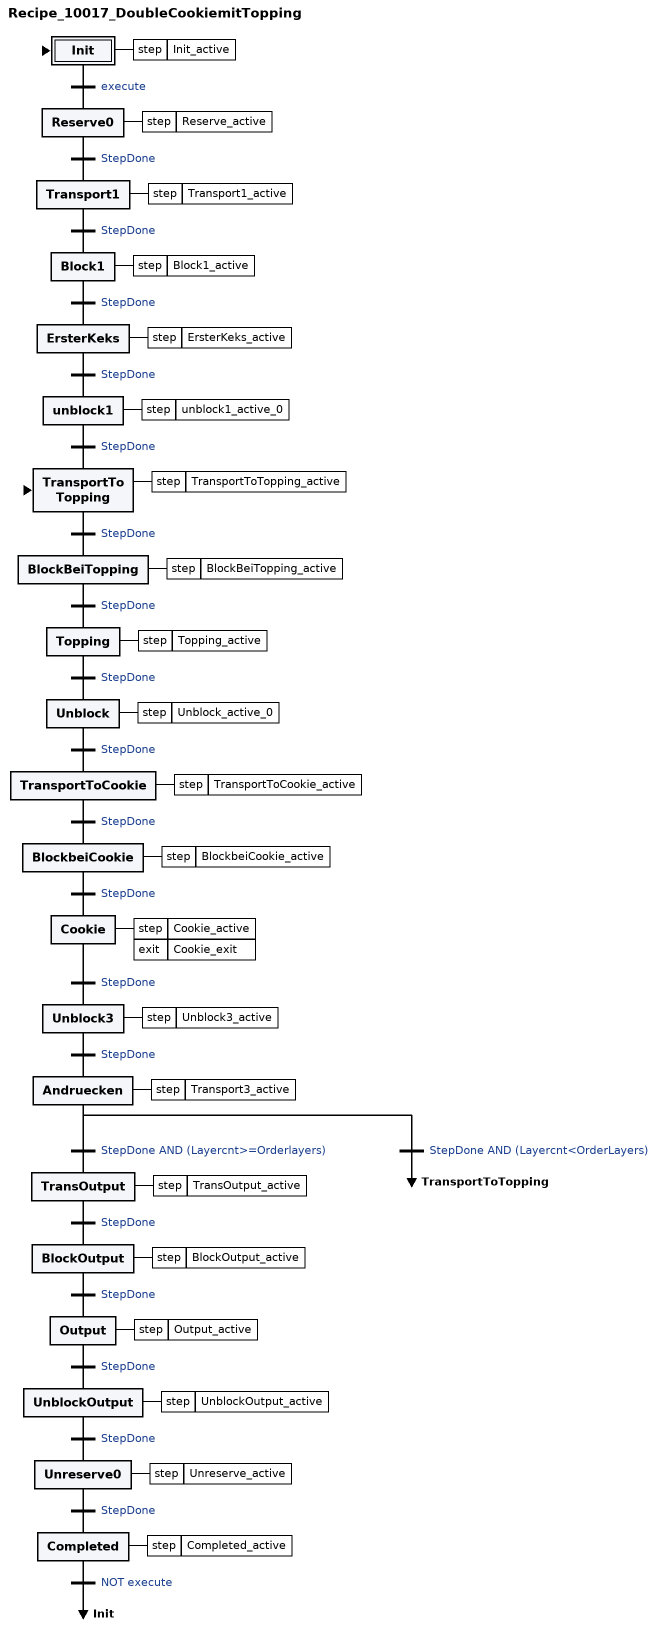
INITIAL_STEP Init:
    Init_active(N);  // step action
END_STEP
TRANSITION FROM Init TO Reserve0
    := execute;
END_TRANSITION
STEP Reserve0:
    Reserve_active(N);  // step action
END_STEP
TRANSITION FROM Reserve0 TO Transport1
    := StepDone;
END_TRANSITION
STEP Transport1:
    Transport1_active(N);  // step action
END_STEP
TRANSITION FROM Transport1 TO Block1
    := StepDone;
END_TRANSITION
STEP Block1:
    Block1_active(N);  // step action
END_STEP
TRANSITION FROM Block1 TO ErsterKeks
    := StepDone;
END_TRANSITION
STEP ErsterKeks:
    ErsterKeks_active(N);  // step action
END_STEP
TRANSITION FROM ErsterKeks TO unblock1
    := StepDone;
END_TRANSITION
STEP unblock1:
    unblock1_active_0(N);  // step action
END_STEP
TRANSITION FROM unblock1 TO TransportToTopping
    := StepDone;
END_TRANSITION
STEP TransportToTopping:
    TransportToTopping_active(N);  // step action
END_STEP
TRANSITION FROM TransportToTopping TO BlockBeiTopping
    := StepDone;
END_TRANSITION
STEP BlockBeiTopping:
    BlockBeiTopping_active(N);  // step action
END_STEP
TRANSITION FROM BlockBeiTopping TO Topping
    := StepDone;
END_TRANSITION
STEP Topping:
    Topping_active(N);  // step action
END_STEP
TRANSITION FROM Topping TO Unblock
    := StepDone;
END_TRANSITION
STEP Unblock:
    Unblock_active_0(N);  // step action
END_STEP
TRANSITION FROM Unblock TO TransportToCookie
    := StepDone;
END_TRANSITION
STEP TransportToCookie:
    TransportToCookie_active(N);  // step action
END_STEP
TRANSITION FROM TransportToCookie TO BlockbeiCookie
    := StepDone;
END_TRANSITION
STEP BlockbeiCookie:
    BlockbeiCookie_active(N);  // step action
END_STEP
TRANSITION FROM BlockbeiCookie TO Cookie
    := StepDone;
END_TRANSITION
STEP Cookie:
    Cookie_active(N);  // step action
    Cookie_exit(P0);  // exit action
END_STEP
TRANSITION FROM Cookie TO Unblock3
    := StepDone;
END_TRANSITION
STEP Unblock3:
    Unblock3_active(N);  // step action
END_STEP
TRANSITION FROM Unblock3 TO Andruecken
    := StepDone;
END_TRANSITION
STEP Andruecken:
    Transport3_active(N);  // step action
END_STEP
TRANSITION FROM Andruecken TO TransOutput
    := StepDone AND (Layercnt>=Orderlayers);
END_TRANSITION
STEP TransOutput:
    TransOutput_active(N);  // step action
END_STEP
TRANSITION FROM TransOutput TO BlockOutput
    := StepDone;
END_TRANSITION
STEP BlockOutput:
    BlockOutput_active(N);  // step action
END_STEP
TRANSITION FROM BlockOutput TO Output
    := StepDone;
END_TRANSITION
STEP Output:
    Output_active(N);  // step action
END_STEP
TRANSITION FROM Output TO UnblockOutput
    := StepDone;
END_TRANSITION
STEP UnblockOutput:
    UnblockOutput_active(N);  // step action
END_STEP
TRANSITION FROM UnblockOutput TO Unreserve0
    := StepDone;
END_TRANSITION
TRANSITION FROM Andruecken TO TransportToTopping
    := StepDone AND (Layercnt<OrderLayers);
END_TRANSITION
STEP Unreserve0:
    Unreserve_active(N);  // step action
END_STEP
TRANSITION FROM Unreserve0 TO Completed
    := StepDone;
END_TRANSITION
STEP Completed:
    Completed_active(N);  // step action
END_STEP
TRANSITION FROM Completed TO Init
    := NOT execute;
END_TRANSITION

ACTION unblock1_active_0:
StepDone := FALSE;

//Skill auswählen
ExecuteSkill.SkillID 		:= 1316;
ExecuteSkill.SkillName	 	:= 'Unblock';

//Parameter setzen

ExecuteSkill.Parameter[1].ID := 1;
ExecuteSkill.Parameter[1].Name := 'TaskID';
ExecuteSkill.Parameter[1].Value := 128 ;


(*
ExecuteSkill.Parameter[2].ID := ;
ExecuteSkill.Parameter[2].Name := '';
ExecuteSkill.Parameter[2].Value := ;
*)

(*
ExecuteSkill.Parameter[3].ID := ;
ExecuteSkill.Parameter[3].Name := '';
ExecuteSkill.Parameter[3].Value := ;
*)

(*
ExecuteSkill.Parameter[4].ID := ;
ExecuteSkill.Parameter[4].Name := '';
ExecuteSkill.Parameter[4].Value := ;
*)

(*
ExecuteSkill.Parameter[5].ID := ;
ExecuteSkill.Parameter[5].Name := '';
ExecuteSkill.Parameter[5].Value := ;
*)



ExecuteSkill();

StepDone := ExecuteSkill.Done;
END_ACTION

ACTION Topping_active:
StepDone := FALSE;

//Skill auswählen
CASE REAL_TO_INT (order.UserParameter[2*LayerCnt].Value) OF
	1: 
		ExecuteSkill.SkillID 		:=  1230;
		ExecuteSkill.SkillName	 	:= 'Strawberry Topping';
	2: 
		ExecuteSkill.SkillID 		:=  1240;
		ExecuteSkill.SkillName	 	:= 'Apple Topping';
	ELSE
		ExecuteSkill.SkillID 		:=  1230;
		ExecuteSkill.SkillName	 	:= 'Strawberry Topping';
END_CASE


//Parameter setzen

ExecuteSkill.Parameter[0].ID := 1;
ExecuteSkill.Parameter[0].Name := 'Amount';
ExecuteSkill.Parameter[0].Value := order.UserParameter[2*LayerCnt + 1].Value ;


(*
ExecuteSkill.Parameter[1].ID := 1;
ExecuteSkill.Parameter[1].Name := 'TaskID';
ExecuteSkill.Parameter[1].Value := 130;
*)
(*
ExecuteSkill.Parameter[2].ID := ;
ExecuteSkill.Parameter[2].Name := '';
ExecuteSkill.Parameter[2].Value := ;
*)

(*
ExecuteSkill.Parameter[3].ID := ;
ExecuteSkill.Parameter[3].Name := '';
ExecuteSkill.Parameter[3].Value := ;
*)

(*
ExecuteSkill.Parameter[4].ID := ;
ExecuteSkill.Parameter[4].Name := '';
ExecuteSkill.Parameter[4].Value := ;
*)

(*
ExecuteSkill.Parameter[5].ID := ;
ExecuteSkill.Parameter[5].Name := '';
ExecuteSkill.Parameter[5].Value := ;
*)

ExecuteSkill();

StepDone := ExecuteSkill.Done;
END_ACTION

ACTION Cookie_active:
StepDone := FALSE;
RecipeDone := FALSE;
//Skill auswählen
ExecuteSkill.SkillID 		:= 1010;
ExecuteSkill.SkillName	 	:= 'Cookie ausgeben';





ExecuteSkill();

StepDone := ExecuteSkill.Done;
END_ACTION

ACTION Transport3_active:
(*StepDone := FALSE;

//Skill auswählen
ExecuteSkill.SkillID 		:= 1320;
ExecuteSkill.SkillName	 	:= 'Transport';

//Parameter setzen

ExecuteSkill.Parameter[3].ID := 3;
ExecuteSkill.Parameter[3].Name := 'Velocity';
ExecuteSkill.Parameter[3].Value := 2800;



ExecuteSkill.Parameter[1].ID :=  1;
ExecuteSkill.Parameter[1].Name := 'TargetPosition X';
ExecuteSkill.Parameter[1].Value := 30 ;
ExecuteSkill.Parameter[1].StringValue := '#DP#-2#XPosition';



ExecuteSkill.Parameter[2].ID := 2;
ExecuteSkill.Parameter[2].Name := 'TargetPosition Z';
ExecuteSkill.Parameter[2].Value := 105;// ZCookieModule - ZCookieModuleCalibration - 2* Cookiethickness + toppingthickness+ Preasureheight  ;



ExecuteSkill.Parameter[4].ID := 4;
ExecuteSkill.Parameter[4].Name := 'Acceleration';
ExecuteSkill.Parameter[4].Value := 2000 ;


(*
ExecuteSkill.Parameter[5].ID := ;
ExecuteSkill.Parameter[5].Name := '';
ExecuteSkill.Parameter[5].Value := ;
*)



ExecuteSkill();

StepDone := ExecuteSkill.Done;
*)
StepDone := TRUE;
END_ACTION

ACTION Completed_active:
RecipeDone := TRUE;
StepDone := FALSE;
Layercnt := 0;
END_ACTION

ACTION BlockbeiCookie_active:
StepDone := FALSE;

//Skill auswählen
ExecuteSkill.SkillID 		:= 1315;
ExecuteSkill.SkillName	 	:= 'Block';

//Parameter setzen

ExecuteSkill.Parameter[1].ID := 1;
ExecuteSkill.Parameter[1].Name := 'TaskID';
ExecuteSkill.Parameter[1].Value := 130;


(*
ExecuteSkill.Parameter[2].ID := ;
ExecuteSkill.Parameter[2].Name := '';
ExecuteSkill.Parameter[2].Value := ;
*)

(*
ExecuteSkill.Parameter[3].ID := ;
ExecuteSkill.Parameter[3].Name := '';
ExecuteSkill.Parameter[3].Value := ;
*)

(*
ExecuteSkill.Parameter[4].ID := ;
ExecuteSkill.Parameter[4].Name := '';
ExecuteSkill.Parameter[4].Value := ;
*)

(*
ExecuteSkill.Parameter[5].ID := ;
ExecuteSkill.Parameter[5].Name := '';
ExecuteSkill.Parameter[5].Value := ;
*)



ExecuteSkill();

StepDone := ExecuteSkill.Done;
END_ACTION

ACTION BlockBeiTopping_active:
StepDone := FALSE;

//Skill auswählen
ExecuteSkill.SkillID 		:= 1315;
ExecuteSkill.SkillName	 	:= 'Block';

//Parameter setzen

ExecuteSkill.Parameter[1].ID := 1;
ExecuteSkill.Parameter[1].Name := 'TaskID';
ExecuteSkill.Parameter[1].Value := 130;


(*
ExecuteSkill.Parameter[2].ID := ;
ExecuteSkill.Parameter[2].Name := '';
ExecuteSkill.Parameter[2].Value := ;
*)

(*
ExecuteSkill.Parameter[3].ID := ;
ExecuteSkill.Parameter[3].Name := '';
ExecuteSkill.Parameter[3].Value := ;
*)

(*
ExecuteSkill.Parameter[4].ID := ;
ExecuteSkill.Parameter[4].Name := '';
ExecuteSkill.Parameter[4].Value := ;
*)

(*
ExecuteSkill.Parameter[5].ID := ;
ExecuteSkill.Parameter[5].Name := '';
ExecuteSkill.Parameter[5].Value := ;
*)



ExecuteSkill();

StepDone := ExecuteSkill.Done;
END_ACTION

ACTION ErsterKeks_active:
StepDone := FALSE;
RecipeDone := FALSE;
//Skill auswählen
ExecuteSkill.SkillID 		:= 1010;
ExecuteSkill.SkillName	 	:= 'Seperate Cookie';


ExecuteSkill();

StepDone := ExecuteSkill.Done;
END_ACTION

ACTION Transport1_active:
StepDone := FALSE;

//Skill auswählen
ExecuteSkill.SkillID 		:= 1320;
ExecuteSkill.SkillName	 	:= 'Transport';

//Parameter setzen

ExecuteSkill.Parameter[3].ID := 3;
ExecuteSkill.Parameter[3].Name := 'Velocity';
ExecuteSkill.Parameter[3].Value := 1500;



ExecuteSkill.Parameter[4].ID := 4 ;
ExecuteSkill.Parameter[4].Name := 'Acceleration';
ExecuteSkill.Parameter[4].Value := 1000 ;



ExecuteSkill.Parameter[1].ID := 1;
ExecuteSkill.Parameter[1].Name := 'TargetPosition X';
ExecuteSkill.Parameter[1].Value := 3200 ;
ExecuteSkill.Parameter[1].StringValue := '#DP#2#XPosition' ;




ExecuteSkill.Parameter[2].ID := 2;
ExecuteSkill.Parameter[2].Name := 'TargetPosition Z';
ExecuteSkill.Parameter[2].Value := ZCookieModule + ZCocktailModuleCalibration;


(*
ExecuteSkill.Parameter[5].ID := ;
ExecuteSkill.Parameter[5].Name := '';
ExecuteSkill.Parameter[5].Value := ;
*)



ExecuteSkill();

StepDone := ExecuteSkill.Done;
END_ACTION

ACTION Production0_active:
StepDone := FALSE;
RecipeDone := FALSE; 
//simulation ausgewählt?
CASE LREAL_TO_INT (order.UserParameter[2].Value) OF

1:
ExecuteSkill.SkillID 		:= 1337;
ExecuteSkill.SkillName	 	:= 'Testskill';

ExecuteSkill();

StepDone := ExecuteSkill.Done;
ELSE StepDone := TRUE;

END_CASE
END_ACTION

ACTION TransportToTopping_active:
StepDone := FALSE;

//Skill auswählen
ExecuteSkill.SkillID 		:= 1320;
ExecuteSkill.SkillName	 	:= 'Transport';

//Parameter setzen

ExecuteSkill.Parameter[3].ID := 3;
ExecuteSkill.Parameter[3].Name := 'Velocity';
ExecuteSkill.Parameter[3].Value := 1000;



ExecuteSkill.Parameter[1].ID :=  1;
ExecuteSkill.Parameter[1].Name := 'TargetPosition X';
ExecuteSkill.Parameter[1].Value := 30 ;
ExecuteSkill.Parameter[1].StringValue := '#DP#2#XPosition';



ExecuteSkill.Parameter[2].ID := 2;
ExecuteSkill.Parameter[2].Name := 'TargetPosition Z';
ExecuteSkill.Parameter[2].Value := ZCremeModule + ZCremeModuleCalibration - Layercnt * ( cookiethickness + toppingthickness);

ExecuteSkill();

StepDone := ExecuteSkill.Done;
END_ACTION

ACTION UnblockOutput_active:
StepDone := FALSE;

//Skill auswählen
ExecuteSkill.SkillID 		:= 1316;
ExecuteSkill.SkillName	 	:= 'Unblock';

//Parameter setzen



(*
ExecuteSkill.Parameter[2].ID := ;
ExecuteSkill.Parameter[2].Name := '';
ExecuteSkill.Parameter[2].Value := ;
*)

(*
ExecuteSkill.Parameter[3].ID := ;
ExecuteSkill.Parameter[3].Name := '';
ExecuteSkill.Parameter[3].Value := ;
*)

(*
ExecuteSkill.Parameter[4].ID := ;
ExecuteSkill.Parameter[4].Name := '';
ExecuteSkill.Parameter[4].Value := ;
*)

(*
ExecuteSkill.Parameter[5].ID := ;
ExecuteSkill.Parameter[5].Name := '';
ExecuteSkill.Parameter[5].Value := ;
*)



ExecuteSkill();

StepDone := ExecuteSkill.Done;
END_ACTION

ACTION BlockOutput_active:
StepDone := FALSE;

//Skill auswählen



ExecuteSkill.SkillID 		:= 1315;
ExecuteSkill.SkillName	 	:= 'Block';

ExecuteSkill();

StepDone := ExecuteSkill.Done;
END_ACTION

ACTION Transport_active:
StepDone := FALSE;

//Skill auswählen

CASE LREAL_TO_INT (order.UserParameter[2].Value) OF

1:
//Skill auswählen
ExecuteSkill.SkillID 		:= 1320;
ExecuteSkill.SkillName	 	:= 'Transport';

//Parameter setzen

ExecuteSkill.Parameter[3].ID :=3 ;
ExecuteSkill.Parameter[3].Name := 'Velocity';
ExecuteSkill.Parameter[3].Value := 1500;



ExecuteSkill.Parameter[1].ID :=1 ;
ExecuteSkill.Parameter[1].Name := 'TargetPosition X';
ExecuteSkill.Parameter[1].StringValue := '#DP#2#XPosition';
ExecuteSkill.Parameter[1].Value := 200 ;


ExecuteSkill.Parameter[2].ID := 2 ;
ExecuteSkill.Parameter[2].Name := 'TargetPosition Z';
ExecuteSkill.Parameter[2].Value := 90 ;



ExecuteSkill.Parameter[4].ID := 4 ;
ExecuteSkill.Parameter[4].Name := 'Acceleration';
ExecuteSkill.Parameter[4].Value := 4500;


(*
ExecuteSkill.Parameter[5].ID := ;
ExecuteSkill.Parameter[5].Name := '';
ExecuteSkill.Parameter[5].Value := ;
*)



ExecuteSkill();

StepDone := ExecuteSkill.Done;
ELSE StepDone := TRUE;

END_CASE
END_ACTION

ACTION Unblock_active:
StepDone := FALSE;

//Skill auswählen
ExecuteSkill.SkillID 		:= 1316;
ExecuteSkill.SkillName	 	:= 'Unblock';

//Parameter setzen

ExecuteSkill.Parameter[1].ID := 1;
ExecuteSkill.Parameter[1].Name := 'TaskID';
ExecuteSkill.Parameter[1].Value := 125;


(*
ExecuteSkill.Parameter[2].ID := ;
ExecuteSkill.Parameter[2].Name := '';
ExecuteSkill.Parameter[2].Value := ;
*)

(*
ExecuteSkill.Parameter[3].ID := ;
ExecuteSkill.Parameter[3].Name := '';
ExecuteSkill.Parameter[3].Value := ;
*)

(*
ExecuteSkill.Parameter[4].ID := ;
ExecuteSkill.Parameter[4].Name := '';
ExecuteSkill.Parameter[4].Value := ;
*)

(*
ExecuteSkill.Parameter[5].ID := ;
ExecuteSkill.Parameter[5].Name := '';
ExecuteSkill.Parameter[5].Value := ;
*)



ExecuteSkill();

StepDone := ExecuteSkill.Done;
END_ACTION

ACTION Production2_active:
StepDone := FALSE;
RecipeDone := FALSE;
//Skill auswählen
ExecuteSkill.SkillID 		:= 1339;
ExecuteSkill.SkillName	 	:= 'ParameterTESTSKILL1339';


ExecuteSkill.Parameter[0].ID := 10;
ExecuteSkill.Parameter[0].Name := 'Blinkfrequenz';
ExecuteSkill.Parameter[0].Value := Order.UserParameter[0].Value*2;


ExecuteSkill();

StepDone := ExecuteSkill.Done;
END_ACTION

ACTION Unblock3_active:
StepDone := FALSE;

//Skill auswählen
ExecuteSkill.SkillID 		:= 1316;
ExecuteSkill.SkillName	 	:= 'Unblock';

//Parameter setzen

